	.N61_OUT AT %QB244 : ST_PSX_VALVE_OUT;	(*  ~ {LinkedWith:TIID^CAN 1 (BOW) ^PSX 61 (MF04)^RxPDO 1^Outputs^Device control word;TIID^CAN 1 (BOW) ^PSX 61 (MF04)^RxPDO 1^Outputs^vpoc_set_point_Value} *)
	.N64_OUT AT %QB248 : ST_PSX_VALVE_OUT;	(*  ~ {LinkedWith:TIID^CAN 1 (BOW) ^PSX 64 (MF04)^RxPDO 1^Outputs^Device control word;TIID^CAN 1 (BOW) ^PSX 64 (MF04)^RxPDO 1^Outputs^vpoc_set_point_Value} *)
	.EV4801 AT %QX696.0 : BOOL;
	.EV4802 AT %QX696.1 : BOOL;
	.EV4803 AT %QX696.2 : BOOL;
	.EV4804 AT %QX696.3 : BOOL;
	.N102_IN AT %IB502 : WORD;	(*  ~ {LinkedWith:TIID^CAN 4 (PANEL)^Box 102 (K-tronic CANopen Cariboni)^TxPDO 1^Entradas^Inputs} *)
	.N103_IN AT %IB504 : WORD;	(*  ~ {LinkedWith:TIID^CAN 4 (PANEL)^Box 103 (K-tronic CANopen Cariboni)^TxPDO 1^Entradas^Inputs} *)
	.N104_IN AT %IB506 : WORD;	(*  ~ {LinkedWith:TIID^CAN 4 (PANEL)^Box 104 (K-tronic CANopen Cariboni)^TxPDO 1^Entradas^Inputs} *)
	.N105_IN AT %IB508 : WORD;	(*  ~ {LinkedWith:TIID^CAN 4 (PANEL)^Box 105 (K-tronic CANopen Cariboni)^TxPDO 1^Entradas^Inputs} *)
	.N106_IN AT %IB510 : WORD;	(*  ~ {LinkedWith:TIID^CAN 4 (PANEL)^Box 106 (K-tronic CANopen Cariboni)^TxPDO 1^Entradas^Inputs} *)
	.N107_IN AT %IB512 : WORD;	(*  ~ {LinkedWith:TIID^CAN 4 (PANEL)^Box 107 (K-tronic CANopen Cariboni)^TxPDO 1^Entradas^Inputs} *)
	.N108_IN AT %IB514 : WORD;	(*  ~ {LinkedWith:TIID^CAN 4 (PANEL)^Box 108 (K-tronic CANopen Cariboni)^TxPDO 1^Entradas^Inputs} *)
	.N109_IN AT %IB516 : WORD;	(*  ~ {LinkedWith:TIID^CAN 4 (PANEL)^Box 109 (K-tronic CANopen Cariboni)^TxPDO 1^Entradas^Inputs} *)
	.N110_IN AT %IB518 : WORD;	(*  ~ {LinkedWith:TIID^CAN 4 (PANEL)^Box 110 (K-tronic CANopen Cariboni)^TxPDO 1^Entradas^Inputs} *)
	.N111_IN AT %IB520 : WORD;	(*  ~ {LinkedWith:TIID^CAN 4 (PANEL)^Box 111 (K-tronic CANopen Cariboni)^TxPDO 1^Entradas^Inputs} *)
	.N112_IN AT %IB522 : WORD;	(*  ~ {LinkedWith:TIID^CAN 4 (PANEL)^Box 112 (K-tronic CANopen Cariboni)^TxPDO 1^Entradas^Inputs} *)
	.N113_IN AT %IB524 : WORD;	(*  ~ {LinkedWith:TIID^CAN 4 (PANEL)^Box 113 (K-tronic CANopen Cariboni)^TxPDO 1^Entradas^Inputs} *)
	.N114_IN AT %IB526 : WORD;	(*  ~ {LinkedWith:TIID^CAN 4 (PANEL)^Box 114 (K-tronic CANopen Cariboni)^TxPDO 1^Entradas^Inputs} *)
	.N115_IN AT %IB528 : WORD;	(*  ~ {LinkedWith:TIID^CAN 4 (PANEL)^Box 115 (K-tronic CANopen Cariboni)^TxPDO 1^Entradas^Inputs} *)
	.N116_IN AT %IB530 : WORD;	(*  ~ {LinkedWith:TIID^CAN 4 (PANEL)^Box 116 (K-tronic CANopen Cariboni)^TxPDO 1^Entradas^Inputs} *)
	.N117_IN AT %IB532 : WORD;	(*  ~ {LinkedWith:TIID^CAN 4 (PANEL)^Box 117 (K-tronic CANopen Cariboni)^TxPDO 1^Entradas^Inputs} *)
	.N118_IN AT %IB534 : WORD;	(*  ~ {LinkedWith:TIID^CAN 4 (PANEL)^Box 118 (K-tronic CANopen Cariboni)^TxPDO 1^Entradas^Inputs} *)
	.N119_IN AT %IB536 : WORD;	(*  ~ {LinkedWith:TIID^CAN 4 (PANEL)^Box 119 (K-tronic CANopen Cariboni)^TxPDO 1^Entradas^Inputs} *)
	.N120_IN AT %IB744 : WORD;	(*  ~ {LinkedWith:TIID^CAN 4 (PANEL)^Box 120 (bLink)^TxPDO 1^Entradas^IN} *)
	.N121_IN AT %IB746 : WORD;	(*  ~ {LinkedWith:TIID^CAN 4 (PANEL)^Box 121 (bLink)^TxPDO 1^Entradas^IN} *)
	.N102_OUT AT %QB252 : WORD;	(*  ~ {LinkedWith:TIID^CAN 4 (PANEL)^Box 102 (K-tronic CANopen Cariboni)^RxPDO 1^Salidas^Outputs} *)
	.N103_OUT AT %QB254 : WORD;	(*  ~ {LinkedWith:TIID^CAN 4 (PANEL)^Box 103 (K-tronic CANopen Cariboni)^RxPDO 1^Salidas^Outputs} *)
	.N104_OUT AT %QB256 : WORD;	(*  ~ {LinkedWith:TIID^CAN 4 (PANEL)^Box 104 (K-tronic CANopen Cariboni)^RxPDO 1^Salidas^Outputs} *)
	.N105_OUT AT %QB258 : WORD;	(*  ~ {LinkedWith:TIID^CAN 4 (PANEL)^Box 105 (K-tronic CANopen Cariboni)^RxPDO 1^Salidas^Outputs} *)
	.N106_OUT AT %QB260 : WORD;	(*  ~ {LinkedWith:TIID^CAN 4 (PANEL)^Box 106 (K-tronic CANopen Cariboni)^RxPDO 1^Salidas^Outputs} *)
	.N107_OUT AT %QB262 : WORD;	(*  ~ {LinkedWith:TIID^CAN 4 (PANEL)^Box 107 (K-tronic CANopen Cariboni)^RxPDO 1^Salidas^Outputs} *)
	.N108_OUT AT %QB264 : WORD;	(*  ~ {LinkedWith:TIID^CAN 4 (PANEL)^Box 108 (K-tronic CANopen Cariboni)^RxPDO 1^Salidas^Outputs} *)
	.N109_OUT AT %QB266 : WORD;	(*  ~ {LinkedWith:TIID^CAN 4 (PANEL)^Box 109 (K-tronic CANopen Cariboni)^RxPDO 1^Salidas^Outputs} *)
	.N110_OUT AT %QB268 : WORD;	(*  ~ {LinkedWith:TIID^CAN 4 (PANEL)^Box 110 (K-tronic CANopen Cariboni)^RxPDO 1^Salidas^Outputs} *)
	.N111_OUT AT %QB270 : WORD;	(*  ~ {LinkedWith:TIID^CAN 4 (PANEL)^Box 111 (K-tronic CANopen Cariboni)^RxPDO 1^Salidas^Outputs} *)
	.N112_OUT AT %QB272 : WORD;	(*  ~ {LinkedWith:TIID^CAN 4 (PANEL)^Box 112 (K-tronic CANopen Cariboni)^RxPDO 1^Salidas^Outputs} *)
	.N113_OUT AT %QB274 : WORD;	(*  ~ {LinkedWith:TIID^CAN 4 (PANEL)^Box 113 (K-tronic CANopen Cariboni)^RxPDO 1^Salidas^Outputs} *)
	.N114_OUT AT %QB276 : WORD;	(*  ~ {LinkedWith:TIID^CAN 4 (PANEL)^Box 114 (K-tronic CANopen Cariboni)^RxPDO 1^Salidas^Outputs} *)
	.N115_OUT AT %QB278 : WORD;	(*  ~ {LinkedWith:TIID^CAN 4 (PANEL)^Box 115 (K-tronic CANopen Cariboni)^RxPDO 1^Salidas^Outputs} *)
	.N116_OUT AT %QB280 : WORD;	(*  ~ {LinkedWith:TIID^CAN 4 (PANEL)^Box 116 (K-tronic CANopen Cariboni)^RxPDO 1^Salidas^Outputs} *)
	.N117_OUT AT %QB282 : WORD;	(*  ~ {LinkedWith:TIID^CAN 4 (PANEL)^Box 117 (K-tronic CANopen Cariboni)^RxPDO 1^Salidas^Outputs} *)
	.N118_OUT AT %QB284 : WORD;	(*  ~ {LinkedWith:TIID^CAN 4 (PANEL)^Box 118 (K-tronic CANopen Cariboni)^RxPDO 1^Salidas^Outputs} *)
	.N119_OUT AT %QB286 : WORD;	(*  ~ {LinkedWith:TIID^CAN 4 (PANEL)^Box 119 (K-tronic CANopen Cariboni)^RxPDO 1^Salidas^Outputs} *)
	.N120_LED_R AT %QB664 : WORD;	(*  ~ {LinkedWith:TIID^CAN 4 (PANEL)^Box 120 (bLink)^RxPDO 1^Salidas^ON_RED} *)
	.N120_LED_G AT %QB666 : WORD;	(*  ~ {LinkedWith:TIID^CAN 4 (PANEL)^Box 120 (bLink)^RxPDO 1^Salidas^ON_GREEN} *)
	.N120_LED_B AT %QB668 : WORD;	(*  ~ {LinkedWith:TIID^CAN 4 (PANEL)^Box 120 (bLink)^RxPDO 1^Salidas^ON_BLUE} *)
	.N121_LED_R AT %QB670 : WORD;	(*  ~ {LinkedWith:TIID^CAN 4 (PANEL)^Box 121 (bLink)^RxPDO 1^Salidas^ON_RED} *)
	.N121_LED_G AT %QB672 : WORD;	(*  ~ {LinkedWith:TIID^CAN 4 (PANEL)^Box 121 (bLink)^RxPDO 1^Salidas^ON_GREEN} *)
	.N121_LED_B AT %QB674 : WORD;	(*  ~ {LinkedWith:TIID^CAN 4 (PANEL)^Box 121 (bLink)^RxPDO 1^Salidas^ON_BLUE} *)
	.N102_BLINK AT %QB288 : WORD;	(*  ~ {LinkedWith:TIID^CAN 4 (PANEL)^Box 102 (K-tronic CANopen Cariboni)^RxPDO 1^Salidas^BlinkOut} *)
	.N103_BLINK AT %QB290 : WORD;	(*  ~ {LinkedWith:TIID^CAN 4 (PANEL)^Box 103 (K-tronic CANopen Cariboni)^RxPDO 1^Salidas^BlinkOut} *)
	.N104_BLINK AT %QB292 : WORD;	(*  ~ {LinkedWith:TIID^CAN 4 (PANEL)^Box 104 (K-tronic CANopen Cariboni)^RxPDO 1^Salidas^BlinkOut} *)
	.N105_BLINK AT %QB294 : WORD;	(*  ~ {LinkedWith:TIID^CAN 4 (PANEL)^Box 105 (K-tronic CANopen Cariboni)^RxPDO 1^Salidas^BlinkOut} *)
	.N106_BLINK AT %QB296 : WORD;	(*  ~ {LinkedWith:TIID^CAN 4 (PANEL)^Box 106 (K-tronic CANopen Cariboni)^RxPDO 1^Salidas^BlinkOut} *)
	.N107_BLINK AT %QB298 : WORD;	(*  ~ {LinkedWith:TIID^CAN 4 (PANEL)^Box 107 (K-tronic CANopen Cariboni)^RxPDO 1^Salidas^BlinkOut} *)
	.N108_BLINK AT %QB300 : WORD;	(*  ~ {LinkedWith:TIID^CAN 4 (PANEL)^Box 108 (K-tronic CANopen Cariboni)^RxPDO 1^Salidas^BlinkOut} *)
	.N109_BLINK AT %QB302 : WORD;	(*  ~ {LinkedWith:TIID^CAN 4 (PANEL)^Box 109 (K-tronic CANopen Cariboni)^RxPDO 1^Salidas^BlinkOut} *)
	.N110_BLINK AT %QB304 : WORD;	(*  ~ {LinkedWith:TIID^CAN 4 (PANEL)^Box 110 (K-tronic CANopen Cariboni)^RxPDO 1^Salidas^BlinkOut} *)
	.N111_BLINK AT %QB306 : WORD;	(*  ~ {LinkedWith:TIID^CAN 4 (PANEL)^Box 111 (K-tronic CANopen Cariboni)^RxPDO 1^Salidas^BlinkOut} *)
	.N112_BLINK AT %QB308 : WORD;	(*  ~ {LinkedWith:TIID^CAN 4 (PANEL)^Box 112 (K-tronic CANopen Cariboni)^RxPDO 1^Salidas^BlinkOut} *)
	.N113_BLINK AT %QB310 : WORD;	(*  ~ {LinkedWith:TIID^CAN 4 (PANEL)^Box 113 (K-tronic CANopen Cariboni)^RxPDO 1^Salidas^BlinkOut} *)
	.N114_BLINK AT %QB312 : WORD;	(*  ~ {LinkedWith:TIID^CAN 4 (PANEL)^Box 114 (K-tronic CANopen Cariboni)^RxPDO 1^Salidas^BlinkOut} *)
	.N115_BLINK AT %QB314 : WORD;	(*  ~ {LinkedWith:TIID^CAN 4 (PANEL)^Box 115 (K-tronic CANopen Cariboni)^RxPDO 1^Salidas^BlinkOut} *)
	.N116_BLINK AT %QB316 : WORD;	(*  ~ {LinkedWith:TIID^CAN 4 (PANEL)^Box 116 (K-tronic CANopen Cariboni)^RxPDO 1^Salidas^BlinkOut} *)
	.N117_BLINK AT %QB318 : WORD;	(*  ~ {LinkedWith:TIID^CAN 4 (PANEL)^Box 117 (K-tronic CANopen Cariboni)^RxPDO 1^Salidas^BlinkOut} *)
	.N118_BLINK AT %QB320 : WORD;	(*  ~ {LinkedWith:TIID^CAN 4 (PANEL)^Box 118 (K-tronic CANopen Cariboni)^RxPDO 1^Salidas^BlinkOut} *)
	.N119_BLINK AT %QB322 : WORD;	(*  ~ {LinkedWith:TIID^CAN 4 (PANEL)^Box 119 (K-tronic CANopen Cariboni)^RxPDO 1^Salidas^BlinkOut} *)
	.N120_BLINK_R AT %QB676 : WORD;	(*  ~ {LinkedWith:TIID^CAN 4 (PANEL)^Box 120 (bLink)^RxPDO 2^Salidas^BLINK_RED} *)
	.N120_BLINK_G AT %QB678 : WORD;	(*  ~ {LinkedWith:TIID^CAN 4 (PANEL)^Box 120 (bLink)^RxPDO 2^Salidas^BLINK_GREEN} *)
	.N120_BLINK_B AT %QB680 : WORD;	(*  ~ {LinkedWith:TIID^CAN 4 (PANEL)^Box 120 (bLink)^RxPDO 2^Salidas^BLINK_BLUE} *)
	.N121_BLINK_R AT %QB682 : WORD;	(*  ~ {LinkedWith:TIID^CAN 4 (PANEL)^Box 121 (bLink)^RxPDO 2^Salidas^BLINK_RED} *)
	.N121_BLINK_G AT %QB684 : WORD;	(*  ~ {LinkedWith:TIID^CAN 4 (PANEL)^Box 121 (bLink)^RxPDO 2^Salidas^BLINK_GREEN} *)
	.N121_BLINK_B AT %QB686 : WORD;	(*  ~ {LinkedWith:TIID^CAN 4 (PANEL)^Box 121 (bLink)^RxPDO 2^Salidas^BLINK_BLUE} *)
	.N102_BTIME AT %QB324 : BYTE;	(*  ~ {LinkedWith:TIID^CAN 4 (PANEL)^Box 102 (K-tronic CANopen Cariboni)^RxPDO 1^Salidas^BlinkTime} *)
	.N103_BTIME AT %QB325 : BYTE;	(*  ~ {LinkedWith:TIID^CAN 4 (PANEL)^Box 103 (K-tronic CANopen Cariboni)^RxPDO 1^Salidas^BlinkTime} *)
	.N104_BTIME AT %QB326 : BYTE;	(*  ~ {LinkedWith:TIID^CAN 4 (PANEL)^Box 104 (K-tronic CANopen Cariboni)^RxPDO 1^Salidas^BlinkTime} *)
	.N105_BTIME AT %QB327 : BYTE;	(*  ~ {LinkedWith:TIID^CAN 4 (PANEL)^Box 105 (K-tronic CANopen Cariboni)^RxPDO 1^Salidas^BlinkTime} *)
	.N106_BTIME AT %QB328 : BYTE;	(*  ~ {LinkedWith:TIID^CAN 4 (PANEL)^Box 106 (K-tronic CANopen Cariboni)^RxPDO 1^Salidas^BlinkTime} *)
	.N107_BTIME AT %QB329 : BYTE;	(*  ~ {LinkedWith:TIID^CAN 4 (PANEL)^Box 107 (K-tronic CANopen Cariboni)^RxPDO 1^Salidas^BlinkTime} *)
	.N108_BTIME AT %QB330 : BYTE;	(*  ~ {LinkedWith:TIID^CAN 4 (PANEL)^Box 108 (K-tronic CANopen Cariboni)^RxPDO 1^Salidas^BlinkTime} *)
	.N109_BTIME AT %QB331 : BYTE;	(*  ~ {LinkedWith:TIID^CAN 4 (PANEL)^Box 109 (K-tronic CANopen Cariboni)^RxPDO 1^Salidas^BlinkTime} *)
	.N110_BTIME AT %QB332 : BYTE;	(*  ~ {LinkedWith:TIID^CAN 4 (PANEL)^Box 110 (K-tronic CANopen Cariboni)^RxPDO 1^Salidas^BlinkTime} *)
	.N111_BTIME AT %QB333 : BYTE;	(*  ~ {LinkedWith:TIID^CAN 4 (PANEL)^Box 111 (K-tronic CANopen Cariboni)^RxPDO 1^Salidas^BlinkTime} *)
	.N112_BTIME AT %QB334 : BYTE;	(*  ~ {LinkedWith:TIID^CAN 4 (PANEL)^Box 112 (K-tronic CANopen Cariboni)^RxPDO 1^Salidas^BlinkTime} *)
	.N113_BTIME AT %QB335 : BYTE;	(*  ~ {LinkedWith:TIID^CAN 4 (PANEL)^Box 113 (K-tronic CANopen Cariboni)^RxPDO 1^Salidas^BlinkTime} *)
	.N114_BTIME AT %QB336 : BYTE;	(*  ~ {LinkedWith:TIID^CAN 4 (PANEL)^Box 114 (K-tronic CANopen Cariboni)^RxPDO 1^Salidas^BlinkTime} *)
	.N115_BTIME AT %QB337 : BYTE;	(*  ~ {LinkedWith:TIID^CAN 4 (PANEL)^Box 115 (K-tronic CANopen Cariboni)^RxPDO 1^Salidas^BlinkTime} *)
	.N116_BTIME AT %QB338 : BYTE;	(*  ~ {LinkedWith:TIID^CAN 4 (PANEL)^Box 116 (K-tronic CANopen Cariboni)^RxPDO 1^Salidas^BlinkTime} *)
	.N117_BTIME AT %QB339 : BYTE;	(*  ~ {LinkedWith:TIID^CAN 4 (PANEL)^Box 117 (K-tronic CANopen Cariboni)^RxPDO 1^Salidas^BlinkTime} *)
	.N118_BTIME AT %QB340 : BYTE;	(*  ~ {LinkedWith:TIID^CAN 4 (PANEL)^Box 118 (K-tronic CANopen Cariboni)^RxPDO 1^Salidas^BlinkTime} *)
	.N119_BTIME AT %QB341 : BYTE;	(*  ~ {LinkedWith:TIID^CAN 4 (PANEL)^Box 119 (K-tronic CANopen Cariboni)^RxPDO 1^Salidas^BlinkTime} *)
	.N102_DIMMER AT %QB342 : WORD;	(*  ~ {LinkedWith:TIID^CAN 4 (PANEL)^Box 102 (K-tronic CANopen Cariboni)^RxPDO 3^Salidas^Dimmer1} *)
	.N103_DIMMER AT %QB344 : WORD;	(*  ~ {LinkedWith:TIID^CAN 4 (PANEL)^Box 103 (K-tronic CANopen Cariboni)^RxPDO 3^Salidas^Dimmer1} *)
	.N104_DIMMER AT %QB346 : WORD;	(*  ~ {LinkedWith:TIID^CAN 4 (PANEL)^Box 104 (K-tronic CANopen Cariboni)^RxPDO 3^Salidas^Dimmer1} *)
	.N105_DIMMER AT %QB348 : WORD;	(*  ~ {LinkedWith:TIID^CAN 4 (PANEL)^Box 105 (K-tronic CANopen Cariboni)^RxPDO 3^Salidas^Dimmer1} *)
	.N106_DIMMER AT %QB350 : WORD;	(*  ~ {LinkedWith:TIID^CAN 4 (PANEL)^Box 106 (K-tronic CANopen Cariboni)^RxPDO 3^Salidas^Dimmer1} *)
	.N107_DIMMER AT %QB352 : WORD;	(*  ~ {LinkedWith:TIID^CAN 4 (PANEL)^Box 107 (K-tronic CANopen Cariboni)^RxPDO 3^Salidas^Dimmer1} *)
	.N108_DIMMER AT %QB354 : WORD;	(*  ~ {LinkedWith:TIID^CAN 4 (PANEL)^Box 108 (K-tronic CANopen Cariboni)^RxPDO 3^Salidas^Dimmer1} *)
	.N109_DIMMER AT %QB356 : WORD;	(*  ~ {LinkedWith:TIID^CAN 4 (PANEL)^Box 109 (K-tronic CANopen Cariboni)^RxPDO 3^Salidas^Dimmer1} *)
	.N110_DIMMER AT %QB358 : WORD;	(*  ~ {LinkedWith:TIID^CAN 4 (PANEL)^Box 110 (K-tronic CANopen Cariboni)^RxPDO 3^Salidas^Dimmer1} *)
	.N111_DIMMER AT %QB360 : WORD;	(*  ~ {LinkedWith:TIID^CAN 4 (PANEL)^Box 111 (K-tronic CANopen Cariboni)^RxPDO 3^Salidas^Dimmer1} *)
	.N112_DIMMER AT %QB362 : WORD;	(*  ~ {LinkedWith:TIID^CAN 4 (PANEL)^Box 112 (K-tronic CANopen Cariboni)^RxPDO 3^Salidas^Dimmer1} *)
	.N113_DIMMER AT %QB364 : WORD;	(*  ~ {LinkedWith:TIID^CAN 4 (PANEL)^Box 113 (K-tronic CANopen Cariboni)^RxPDO 3^Salidas^Dimmer1} *)
	.N114_DIMMER AT %QB366 : WORD;	(*  ~ {LinkedWith:TIID^CAN 4 (PANEL)^Box 114 (K-tronic CANopen Cariboni)^RxPDO 3^Salidas^Dimmer1} *)
	.N115_DIMMER AT %QB368 : WORD;	(*  ~ {LinkedWith:TIID^CAN 4 (PANEL)^Box 115 (K-tronic CANopen Cariboni)^RxPDO 3^Salidas^Dimmer1} *)
	.N116_DIMMER AT %QB370 : WORD;	(*  ~ {LinkedWith:TIID^CAN 4 (PANEL)^Box 116 (K-tronic CANopen Cariboni)^RxPDO 3^Salidas^Dimmer1} *)
	.N117_DIMMER AT %QB372 : WORD;	(*  ~ {LinkedWith:TIID^CAN 4 (PANEL)^Box 117 (K-tronic CANopen Cariboni)^RxPDO 3^Salidas^Dimmer1} *)
	.N118_DIMMER AT %QB374 : WORD;	(*  ~ {LinkedWith:TIID^CAN 4 (PANEL)^Box 118 (K-tronic CANopen Cariboni)^RxPDO 3^Salidas^Dimmer1} *)
	.N119_DIMMER AT %QB376 : WORD;	(*  ~ {LinkedWith:TIID^CAN 4 (PANEL)^Box 119 (K-tronic CANopen Cariboni)^RxPDO 3^Salidas^Dimmer1} *)
	.N120_LED_Bright AT %QB688 : BYTE;	(*  ~ {LinkedWith:TIID^CAN 4 (PANEL)^Box 120 (bLink)^RxPDO 3^Salidas^LED_BRIGHT} *)
	.N121_LED_Bright AT %QB689 : BYTE;	(*  ~ {LinkedWith:TIID^CAN 4 (PANEL)^Box 121 (bLink)^RxPDO 3^Salidas^LED_BRIGHT} *)
	.N120_BL_Bright AT %QB690 : BYTE;	(*  ~ {LinkedWith:TIID^CAN 4 (PANEL)^Box 120 (bLink)^RxPDO 4^Salidas^BL_BRIGHT} *)
	.N121_BL_Bright AT %QB691 : BYTE;	(*  ~ {LinkedWith:TIID^CAN 4 (PANEL)^Box 121 (bLink)^RxPDO 4^Salidas^BL_BRIGHT} *)
	.N120_BL_Color AT %QB692 : BYTE;	(*  ~ {LinkedWith:TIID^CAN 4 (PANEL)^Box 120 (bLink)^RxPDO 4^Salidas^BL_COLOR} *)
	.N121_BL_Color AT %QB693 : BYTE;	(*  ~ {LinkedWith:TIID^CAN 4 (PANEL)^Box 121 (bLink)^RxPDO 4^Salidas^BL_COLOR} *)
	.CLM8_LED1 AT %QB520 : BYTE;	(*  ~ {LinkedWith:TIID^CAN 4 (PANEL)^Box 10 (CLM8)^COB 0x20A^Salidas^LED} *)
	.CLM8_LED2 AT %QB521 : BYTE;	(*  ~ {LinkedWith:TIID^CAN 4 (PANEL)^Box 10 (CLM8)^COB 0x20B^Salidas^LED} *)
	.CLM8_COLOR1 AT %QB524 : UDINT;	(*  ~ {LinkedWith:TIID^CAN 4 (PANEL)^Box 10 (CLM8)^COB 0x20A^Salidas^COLORS} *)
	.CLM8_COLOR2 AT %QB528 : UDINT;	(*  ~ {LinkedWith:TIID^CAN 4 (PANEL)^Box 10 (CLM8)^COB 0x20B^Salidas^COLORS} *)
	.CLM8_BRIGHT AT %QB532 : BYTE;	(*  ~ {LinkedWith:TIID^CAN 4 (PANEL)^Box 10 (CLM8)^COB 0x72F^Salidas^Brightness} *)
	.N10_DI0 AT %IX768.0 : BOOL;	(*  ~ {LinkedWith:TIID^CAN 5 (EL6751)^N10 (IP1001-510)^Term 1^Channel 1^Input} *)
	.N10_DI1 AT %IX768.1 : BOOL;	(*  ~ {LinkedWith:TIID^CAN 5 (EL6751)^N10 (IP1001-510)^Term 1^Channel 2^Input} *)
	.N10_DI2 AT %IX768.2 : BOOL;	(*  ~ {LinkedWith:TIID^CAN 5 (EL6751)^N10 (IP1001-510)^Term 1^Channel 3^Input} *)
	.N10_DI3 AT %IX768.3 : BOOL;	(*  ~ {LinkedWith:TIID^CAN 5 (EL6751)^N10 (IP1001-510)^Term 1^Channel 4^Input} *)
	.N10_DI4 AT %IX768.4 : BOOL;	(*  ~ {LinkedWith:TIID^CAN 5 (EL6751)^N10 (IP1001-510)^Term 1^Channel 5^Input} *)
	.N10_DI5 AT %IX768.5 : BOOL;	(*  ~ {LinkedWith:TIID^CAN 5 (EL6751)^N10 (IP1001-510)^Term 1^Channel 6^Input} *)
	.N10_DI6 AT %IX768.6 : BOOL;	(*  ~ {LinkedWith:TIID^CAN 5 (EL6751)^N10 (IP1001-510)^Term 1^Channel 7^Input} *)
	.N10_DI7 AT %IX768.7 : BOOL;	(*  ~ {LinkedWith:TIID^CAN 5 (EL6751)^N10 (IP1001-510)^Term 1^Channel 8^Input} *)
	.N11_DI0 AT %IX769.0 : BOOL;	(*  ~ {LinkedWith:TIID^CAN 5 (EL6751)^N11 (IP1001-510)^Term 1^Channel 1^Input} *)
	.N11_DI1 AT %IX769.1 : BOOL;	(*  ~ {LinkedWith:TIID^CAN 5 (EL6751)^N11 (IP1001-510)^Term 1^Channel 2^Input} *)
	.N11_DI2 AT %IX769.2 : BOOL;	(*  ~ {LinkedWith:TIID^CAN 5 (EL6751)^N11 (IP1001-510)^Term 1^Channel 3^Input} *)
	.N11_DI3 AT %IX769.3 : BOOL;	(*  ~ {LinkedWith:TIID^CAN 5 (EL6751)^N11 (IP1001-510)^Term 1^Channel 4^Input} *)
	.N11_DI4 AT %IX769.4 : BOOL;	(*  ~ {LinkedWith:TIID^CAN 5 (EL6751)^N11 (IP1001-510)^Term 1^Channel 5^Input} *)
	.N11_DI5 AT %IX769.5 : BOOL;	(*  ~ {LinkedWith:TIID^CAN 5 (EL6751)^N11 (IP1001-510)^Term 1^Channel 6^Input} *)
	.N11_DI6 AT %IX769.6 : BOOL;	(*  ~ {LinkedWith:TIID^CAN 5 (EL6751)^N11 (IP1001-510)^Term 1^Channel 7^Input} *)
	.N11_DI7 AT %IX769.7 : BOOL;	(*  ~ {LinkedWith:TIID^CAN 5 (EL6751)^N11 (IP1001-510)^Term 1^Channel 8^Input} *)
	.N12_DI0 AT %IX770.0 : BOOL;	(*  ~ {LinkedWith:TIID^CAN 5 (EL6751)^N12 (IP1001-510)^Term 1^Channel 1^Input} *)
	.N12_DI1 AT %IX770.1 : BOOL;	(*  ~ {LinkedWith:TIID^CAN 5 (EL6751)^N12 (IP1001-510)^Term 1^Channel 2^Input} *)
	.N12_DI2 AT %IX770.2 : BOOL;	(*  ~ {LinkedWith:TIID^CAN 5 (EL6751)^N12 (IP1001-510)^Term 1^Channel 3^Input} *)
	.N12_DI3 AT %IX770.3 : BOOL;	(*  ~ {LinkedWith:TIID^CAN 5 (EL6751)^N12 (IP1001-510)^Term 1^Channel 4^Input} *)
	.N12_DI4 AT %IX770.4 : BOOL;	(*  ~ {LinkedWith:TIID^CAN 5 (EL6751)^N12 (IP1001-510)^Term 1^Channel 5^Input} *)
	.N12_DI5 AT %IX770.5 : BOOL;	(*  ~ {LinkedWith:TIID^CAN 5 (EL6751)^N12 (IP1001-510)^Term 1^Channel 6^Input} *)
	.N12_DI6 AT %IX770.6 : BOOL;	(*  ~ {LinkedWith:TIID^CAN 5 (EL6751)^N12 (IP1001-510)^Term 1^Channel 7^Input} *)
	.N12_DI7 AT %IX770.7 : BOOL;	(*  ~ {LinkedWith:TIID^CAN 5 (EL6751)^N12 (IP1001-510)^Term 1^Channel 8^Input} *)
	.N13_DI0 AT %IX771.0 : BOOL;	(*  ~ {LinkedWith:TIID^CAN 5 (EL6751)^N13 (IP1001-510)^Term 1^Channel 1^Input} *)
	.N13_DI1 AT %IX771.1 : BOOL;	(*  ~ {LinkedWith:TIID^CAN 5 (EL6751)^N13 (IP1001-510)^Term 1^Channel 2^Input} *)
	.N13_DI2 AT %IX771.2 : BOOL;	(*  ~ {LinkedWith:TIID^CAN 5 (EL6751)^N13 (IP1001-510)^Term 1^Channel 3^Input} *)
	.N13_DI3 AT %IX771.3 : BOOL;	(*  ~ {LinkedWith:TIID^CAN 5 (EL6751)^N13 (IP1001-510)^Term 1^Channel 4^Input} *)
	.N13_DI4 AT %IX771.4 : BOOL;	(*  ~ {LinkedWith:TIID^CAN 5 (EL6751)^N13 (IP1001-510)^Term 1^Channel 5^Input} *)
	.N13_DI5 AT %IX771.5 : BOOL;	(*  ~ {LinkedWith:TIID^CAN 5 (EL6751)^N13 (IP1001-510)^Term 1^Channel 6^Input} *)
	.N13_DI6 AT %IX771.6 : BOOL;	(*  ~ {LinkedWith:TIID^CAN 5 (EL6751)^N13 (IP1001-510)^Term 1^Channel 7^Input} *)
	.N13_DI7 AT %IX771.7 : BOOL;	(*  ~ {LinkedWith:TIID^CAN 5 (EL6751)^N13 (IP1001-510)^Term 1^Channel 8^Input} *)
	.N20_DI0 AT %IX772.0 : BOOL;	(*  ~ {LinkedWith:TIID^CAN 5 (EL6751)^N20 (IP1001-510)^Term 1^Channel 1^Input} *)
	.N20_DI1 AT %IX772.1 : BOOL;	(*  ~ {LinkedWith:TIID^CAN 5 (EL6751)^N20 (IP1001-510)^Term 1^Channel 2^Input} *)
	.N20_DI2 AT %IX772.2 : BOOL;	(*  ~ {LinkedWith:TIID^CAN 5 (EL6751)^N20 (IP1001-510)^Term 1^Channel 3^Input} *)
	.N20_DI3 AT %IX772.3 : BOOL;	(*  ~ {LinkedWith:TIID^CAN 5 (EL6751)^N20 (IP1001-510)^Term 1^Channel 4^Input} *)
	.N20_DI4 AT %IX772.4 : BOOL;	(*  ~ {LinkedWith:TIID^CAN 5 (EL6751)^N20 (IP1001-510)^Term 1^Channel 5^Input} *)
	.N20_DI5 AT %IX772.5 : BOOL;	(*  ~ {LinkedWith:TIID^CAN 5 (EL6751)^N20 (IP1001-510)^Term 1^Channel 6^Input} *)
	.N20_DI6 AT %IX772.6 : BOOL;	(*  ~ {LinkedWith:TIID^CAN 5 (EL6751)^N20 (IP1001-510)^Term 1^Channel 7^Input} *)
	.N20_DI7 AT %IX772.7 : BOOL;	(*  ~ {LinkedWith:TIID^CAN 5 (EL6751)^N20 (IP1001-510)^Term 1^Channel 8^Input} *)
	.N20_NodeState AT %IB592 : USINT;	(*  ~ {LinkedWith:TIID^CAN 1 (BOW) ^Box 20 (MF06)^Entradas^NodeState} *)
	.N21_NodeState AT %IB593 : USINT;	(*  ~ {LinkedWith:TIID^CAN 1 (BOW) ^Box 21 (MF07/MF11)^Entradas^NodeState} *)
	.N22_NodeState AT %IB594 : USINT;	(*  ~ {LinkedWith:TIID^CAN 1 (BOW) ^Box 22 (MF07)^Entradas^NodeState} *)
	.N23_NodeState AT %IB595 : USINT;	(*  ~ {LinkedWith:TIID^CAN 2 (STERN)^Box 23 (MF08)^Entradas^NodeState} *)
	.N24_NodeState AT %IB596 : USINT;	(*  ~ {LinkedWith:TIID^CAN 2 (STERN)^Box 24 (MF12A)^Entradas^NodeState} *)
	.N25_NodeState AT %IB597 : USINT;	(*  ~ {LinkedWith:TIID^CAN 2 (STERN)^Box 25 (MF12B)^Entradas^NodeState} *)
	.N26_NodeState AT %IB598 : USINT;	(*  ~ {LinkedWith:TIID^CAN 2 (STERN)^Box 26 (MF25)^Entradas^NodeState} *)
	.N27_NodeState AT %IB599 : USINT;	(*  ~ {LinkedWith:TIID^CAN 2 (STERN)^Box 27 (MF22)^Entradas^NodeState} *)
	.N28_NodeState AT %IB600 : USINT;	(*  ~ {LinkedWith:TIID^CAN 2 (STERN)^Box 28 (MF21)^Entradas^NodeState} *)
	.N29_NodeState AT %IB601 : USINT;	(*  ~ {LinkedWith:TIID^CAN 2 (STERN)^Box 29 (MF24)^Entradas^NodeState} *)
	.N30_NodeState AT %IB602 : USINT;	(*  ~ {LinkedWith:TIID^CAN 2 (STERN)^Box 30 (MF23)^Entradas^NodeState} *)
	.N31_NodeState AT %IB603 : USINT;	(*  ~ {LinkedWith:TIID^CAN 2 (STERN)^Box 31 (MF20)^Entradas^NodeState} *)
	.N32_NodeState AT %IB604 : USINT;	(*  ~ {LinkedWith:TIID^CAN 2 (STERN)^Box 32 (MF19)^Entradas^NodeState} *)
	.N33_NodeState AT %IB605 : USINT;	(*  ~ {LinkedWith:TIID^CAN 2 (STERN)^Box 33 (MF13 Traveller)^Entradas^NodeState} *)
	.N34_NodeState AT %IB606 : USINT;	(*  ~ {LinkedWith:TIID^CAN 2 (STERN)^Box 34 (MF16)^Entradas^NodeState} *)
	.N35_NodeState AT %IB607 : USINT;	(*  ~ {LinkedWith:TIID^CAN 2 (STERN)^Box 35 (MF09)^Entradas^NodeState} *)
	.N36_NodeState AT %IB608 : USINT;	(*  ~ {LinkedWith:TIID^CAN 1 (BOW) ^Box 36 (Tank)^Entradas^NodeState} *)
	.N37_NodeState AT %IB609 : USINT;	(*  ~ {LinkedWith:TIID^CAN 1 (BOW) ^Box 37 (Tank)^Entradas^NodeState} *)
	.N38_NodeState AT %IB610 : USINT;	(*  ~ {LinkedWith:TIID^CAN 2 (STERN)^Box 38 (LIGHT)^Entradas^NodeState} *)
	.N39_NodeState AT %IB611 : USINT;	(*  ~ {LinkedWith:TIID^CAN 1 (BOW) ^Box 39 (MF10A Keel)^Entradas^NodeState} *)
	.N40_NodeState AT %IB612 : USINT;	(*  ~ {LinkedWith:TIID^CAN 1 (BOW) ^Box 40 (MF10B Keel)^Entradas^NodeState} *)
	.N41_NodeState AT %IB613 : USINT;	(*  ~ {LinkedWith:TIID^CAN 1 (BOW) ^Box 41 (MF05)^Entradas^NodeState} *)
	.N42_NodeState AT %IB614 : USINT;	(*  ~ {LinkedWith:TIID^CAN 1 (BOW) ^Box 42 (MF01 HP PP)^Entradas^NodeState} *)
	.N43_NodeState AT %IB615 : USINT;	(*  ~ {LinkedWith:TIID^CAN 1 (BOW) ^Box 43 (MF03A)^Entradas^NodeState} *)
	.N44_NodeState AT %IB616 : USINT;	(*  ~ {LinkedWith:TIID^CAN 1 (BOW) ^Box 44 (MF03B)^Entradas^NodeState} *)
	.N47_NodeState AT %IB706 : USINT;	(*  ~ {LinkedWith:TIID^CAN 2 (STERN)^Box 47 (MF11)^Entradas^NodeState} *)
	.N48_NodeState AT %IB764 : USINT;	(*  ~ {LinkedWith:TIID^CAN 1 (BOW) ^Box 48 (DGB Seal)^Entradas^NodeState} *)
	.N50_NodeState AT %IB617 : USINT;	(*  ~ {LinkedWith:TIID^CAN 2 (STERN)^PSX 50 (MF12)^Inputs^NodeState} *)
	.N51_NodeState AT %IB618 : USINT;	(*  ~ {LinkedWith:TIID^CAN 2 (STERN)^PSX 51 (MF12)^Inputs^NodeState} *)
	.N52_NodeState AT %IB619 : USINT;	(*  ~ {LinkedWith:TIID^CAN 2 (STERN)^PSX 52 (MF12)^Inputs^NodeState} *)
	.N53_NodeState AT %IB620 : USINT;	(*  ~ {LinkedWith:TIID^CAN 2 (STERN)^PSX 53 (MF12)^Inputs^NodeState} *)
	.N54_NodeState AT %IB621 : USINT;	(*  ~ {LinkedWith:TIID^CAN 2 (STERN)^PSX 54 (MF12)^Inputs^NodeState} *)
	.N55_NodeState AT %IB622 : USINT;	(*  ~ {LinkedWith:TIID^CAN 2 (STERN)^PSX 55 (MF12)^Inputs^NodeState} *)
	.N56_NodeState AT %IB623 : USINT;	(*  ~ {LinkedWith:TIID^CAN 2 (STERN)^PSX 56 (MF12)^Inputs^NodeState} *)
	.N57_NodeState AT %IB624 : USINT;	(*  ~ {LinkedWith:TIID^CAN 2 (STERN)^PSX 57 (MF12)^Inputs^NodeState} *)
	.N58_NodeState AT %IB625 : USINT;	(*  ~ {LinkedWith:TIID^CAN 2 (STERN)^PSX 58 (MF12)^Inputs^NodeState} *)
	.N59_NodeState AT %IB626 : USINT;	(*  ~ {LinkedWith:TIID^CAN 2 (STERN)^PSX 59 (MF12)^Inputs^NodeState} *)
	.N60_NodeState AT %IB627 : USINT;	(*  ~ {LinkedWith:TIID^CAN 1 (BOW) ^PSX 60 (MF04)^Inputs^NodeState} *)
	.N61_NodeState AT %IB628 : USINT;	(*  ~ {LinkedWith:TIID^CAN 1 (BOW) ^PSX 61 (MF04)^Inputs^NodeState} *)
	.N64_NodeState AT %IB629 : USINT;	(*  ~ {LinkedWith:TIID^CAN 1 (BOW) ^PSX 64 (MF04)^Inputs^NodeState} *)
	.N70_NodeState AT %IB630 : USINT;	(*  ~ {LinkedWith:TIID^CAN 2 (STERN)^PSX 70 (MF16)^Inputs^NodeState} *)
	.N71_NodeState AT %IB631 : USINT;	(*  ~ {LinkedWith:TIID^CAN 2 (STERN)^PSX 71 (MF16)^Inputs^NodeState} *)
	.N72_NodeState AT %IB632 : USINT;	(*  ~ {LinkedWith:TIID^CAN 2 (STERN)^PSX 72 (MF16)^Inputs^NodeState} *)
	.N73_NodeState AT %IB633 : USINT;	(*  ~ {LinkedWith:TIID^CAN 2 (STERN)^PSX 73 (MF16)^Inputs^NodeState} *)
	.N74_NodeState AT %IB634 : USINT;	(*  ~ {LinkedWith:TIID^CAN 2 (STERN)^PSX 74 (MF16)^Inputs^NodeState} *)
	.N102_NodeState AT %IB635 : USINT;	(*  ~ {LinkedWith:TIID^CAN 4 (PANEL)^Box 102 (K-tronic CANopen Cariboni)^Entradas^NodeState} *)
	.N103_NodeState AT %IB636 : USINT;	(*  ~ {LinkedWith:TIID^CAN 4 (PANEL)^Box 103 (K-tronic CANopen Cariboni)^Entradas^NodeState} *)
	.N104_NodeState AT %IB637 : USINT;	(*  ~ {LinkedWith:TIID^CAN 4 (PANEL)^Box 104 (K-tronic CANopen Cariboni)^Entradas^NodeState} *)
	.N105_NodeState AT %IB638 : USINT;	(*  ~ {LinkedWith:TIID^CAN 4 (PANEL)^Box 105 (K-tronic CANopen Cariboni)^Entradas^NodeState} *)
	.N106_NodeState AT %IB639 : USINT;	(*  ~ {LinkedWith:TIID^CAN 4 (PANEL)^Box 106 (K-tronic CANopen Cariboni)^Entradas^NodeState} *)
	.N107_NodeState AT %IB640 : USINT;	(*  ~ {LinkedWith:TIID^CAN 4 (PANEL)^Box 107 (K-tronic CANopen Cariboni)^Entradas^NodeState} *)
	.N108_NodeState AT %IB641 : USINT;	(*  ~ {LinkedWith:TIID^CAN 4 (PANEL)^Box 108 (K-tronic CANopen Cariboni)^Entradas^NodeState} *)
	.N109_NodeState AT %IB642 : USINT;	(*  ~ {LinkedWith:TIID^CAN 4 (PANEL)^Box 109 (K-tronic CANopen Cariboni)^Entradas^NodeState} *)
	.N110_NodeState AT %IB643 : USINT;	(*  ~ {LinkedWith:TIID^CAN 4 (PANEL)^Box 110 (K-tronic CANopen Cariboni)^Entradas^NodeState} *)
	.N111_NodeState AT %IB644 : USINT;	(*  ~ {LinkedWith:TIID^CAN 4 (PANEL)^Box 111 (K-tronic CANopen Cariboni)^Entradas^NodeState} *)
	.N112_NodeState AT %IB645 : USINT;	(*  ~ {LinkedWith:TIID^CAN 4 (PANEL)^Box 112 (K-tronic CANopen Cariboni)^Entradas^NodeState} *)
	.N113_NodeState AT %IB646 : USINT;	(*  ~ {LinkedWith:TIID^CAN 4 (PANEL)^Box 113 (K-tronic CANopen Cariboni)^Entradas^NodeState} *)
	.N114_NodeState AT %IB647 : USINT;	(*  ~ {LinkedWith:TIID^CAN 4 (PANEL)^Box 114 (K-tronic CANopen Cariboni)^Entradas^NodeState} *)
	.N115_NodeState AT %IB648 : USINT;	(*  ~ {LinkedWith:TIID^CAN 4 (PANEL)^Box 115 (K-tronic CANopen Cariboni)^Entradas^NodeState} *)
	.N116_NodeState AT %IB649 : USINT;	(*  ~ {LinkedWith:TIID^CAN 4 (PANEL)^Box 116 (K-tronic CANopen Cariboni)^Entradas^NodeState} *)
	.N117_NodeState AT %IB650 : USINT;	(*  ~ {LinkedWith:TIID^CAN 4 (PANEL)^Box 117 (K-tronic CANopen Cariboni)^Entradas^NodeState} *)
	.N118_NodeState AT %IB651 : USINT;	(*  ~ {LinkedWith:TIID^CAN 4 (PANEL)^Box 118 (K-tronic CANopen Cariboni)^Entradas^NodeState} *)
	.N119_NodeState AT %IB652 : USINT;	(*  ~ {LinkedWith:TIID^CAN 4 (PANEL)^Box 119 (K-tronic CANopen Cariboni)^Entradas^NodeState} *)
	.N120_NodeState AT %IB748 : USINT;	(*  ~ {LinkedWith:TIID^CAN 4 (PANEL)^Box 120 (bLink)^Entradas^NodeState} *)
	.N121_NodeState AT %IB749 : USINT;	(*  ~ {LinkedWith:TIID^CAN 4 (PANEL)^Box 121 (bLink)^Entradas^NodeState} *)
	.N10_NodeState AT %IB661 : USINT;	(*  ~ {LinkedWith:TIID^CAN 5 (EL6751)^N10 (IP1001-510)^Inputs^NodeState} *)
	.N11_NodeState AT %IB662 : USINT;	(*  ~ {LinkedWith:TIID^CAN 5 (EL6751)^N11 (IP1001-510)^Inputs^NodeState} *)
	.N12_NodeState AT %IB663 : USINT;	(*  ~ {LinkedWith:TIID^CAN 5 (EL6751)^N12 (IP1001-510)^Inputs^NodeState} *)
	.N13_NodeState AT %IB664 : USINT;	(*  ~ {LinkedWith:TIID^CAN 5 (EL6751)^N13 (IP1001-510)^Inputs^NodeState} *)
	.N20_2_NodeState AT %IB724 : USINT;	(*  ~ {LinkedWith:TIID^CAN 5 (EL6751)^N20 (IP1001-510)^Inputs^NodeState} *)
END_VAR

(* Data type *)
TYPE RxQueue_10 :
STRUCT
	TxCounter      : UINT;
	RxCounter      : UINT;
	NoOfRxMessages : UINT;
	RxMessages     : ARRAY [0..9] OF ARRAY[0..13] OF BYTE;
END_STRUCT
END_TYPE

(* Data type *)
TYPE ST_ALARM :
STRUCT
	AlLen  : REAL;
	AlCnt  : WORD;
	TimeInit : STRING;
	TimeEnd  : STRING;

	Alarm  : BOOL;
	Adver  : BOOL;
	Text   : STRING;

	AlInit : BOOL;
	AlEnd  : BOOL;
END_STRUCT
END_TYPE

(* Data type *)
TYPE ST_BOARD_CFG :
STRUCT
(*Targets*)
	TgtLS_P_In   : REAL;
	TgtLS_P_InR  : REAL;
	TgtLS_P_Mid  : REAL;
	TgtLS_P_OutR : REAL;
	TgtLS_P_Out  : REAL;

	TgtLS_S_In   : REAL;
	TgtLS_S_InR  : REAL;
	TgtLS_S_Mid  : REAL;
	TgtLS_S_OutR : REAL;
	TgtLS_S_Out  : REAL;

	TgtLS_P_Safe_Out : REAL;
	TgtLS_P_Safe_In  : REAL;

	TgtLS_S_Safe_Out : REAL;
	TgtLS_S_Safe_In  : REAL;

	LS_Dif_Tgt : REAL;
	LS_Dif_Max : REAL;
	LS_Dif_Min : REAL;

	LS_DB : REAL;

	P_Hyst_HP : REAL;
	P_Hyst_LP : REAL;
	P_Hyst_TM : REAL;	(*Seconds*)

(*Keel Limits*)
	Keel_P_Max : REAL;
	Keel_S_Min : REAL;

(*Valve Limits*)
	EVP_In_P_Min  : REAL;
	EVP_In_P_Max  : REAL;

	EVP_In_S_Min  : REAL;
	EVP_In_S_Max  : REAL;

	EVP_Out_P_Min  : REAL;
	EVP_Out_P_Max  : REAL;

	EVP_Out_S_Min  : REAL;
	EVP_Out_S_Max  : REAL;

(*Valve Targets*)
	EVP_In_P_Eng : REAL;
	EVP_In_P_PP  : REAL;

	EVP_In_S_Eng : REAL;
	EVP_In_S_PP  : REAL;

	EVP_Out_P_Eng : REAL;
	EVP_Out_P_PP  : REAL;

	EVP_Out_S_Eng : REAL;
	EVP_Out_S_PP  : REAL;

(*Valve Gains*)
	EVP_In_EVP_K  : REAL;
	EVP_Out_EVP_K : REAL;

	EVP_In_LS_K  : REAL;
	EVP_Out_LS_K : REAL;

(*Valve Softstart*)
	EVP_In_Inc  : REAL;
	EVP_Out_Inc : REAL;

	EVP_In_Dec  : REAL;
	EVP_Out_Dec : REAL;

	LP : BYTE;

	Cycle    : REAL; (*Seconds*)
	TimeMax  : REAL; (*Seconds*)

END_STRUCT
END_TYPE

(* Data type *)
TYPE ST_CAN_NODESTATE :
STRUCT
	Desc : STRING;

	(*Alarm*)
	Alarm  : ST_ALARM;

END_STRUCT
END_TYPE

(* Data type *)
TYPE ST_DE_CYLINDER_POS_CFG :
STRUCT
	TgtLS_In  : REAL;
	TgtLS_Out : REAL;
	TgtLS_Mid : REAL;
	TgtLS_DB  : REAL;

	LS_Limit_In  : BOOL;
	LS_Limit_Out : BOOL;

	Cycle   : REAL; (*Seconds*)
	TimeMax : REAL; (*Seconds*)

	HP : BYTE;
END_STRUCT
END_TYPE

(* Data type *)
TYPE ST_ENGINE_CFG :
STRUCT

	(*Parameters*)
	MaxInc_RPM : REAL; (*RPM/sec*)
	MaxDec_RPM : REAL; (*RPM/sec*)
	DlyDec_sec : REAL;

	Boost_RPM : REAL;
	Max_RPM   : REAL;
	Min_RPM   : REAL;
	Stop_RPM  : REAL;

	HP_Nx_RPM : REAL;
	HP_SF_RPM : REAL;

	LP_CK_RPM : REAL;
	LP_1x_RPM : REAL;
	LP_2x_RPM : REAL;
	LP_3x_RPM : REAL;
	LP_Nx_RPM : REAL;

	N_Winch_WOP : INT;
	N_Winch_WK  : INT;
	N_Winch_WP  : INT;

	Max_Torque : REAL;
	Min_Torque : REAL;

	Inc_RMP_Perc_WOP : REAL;
	Dec_Flow_Perc_WP : REAL;

	Max_HeatExch_P : REAL;

	Cycle : REAL; (*Seconds*)

	EnForceRPM : BOOL;
	EnForceTHR : BOOL;



	(*Coefficients*)
	CycleMaxInc_RPM : REAL;
	CycleMaxDec_RPM : REAL;

	Boost_K : REAL;
	OffDelay_cycl : UINT;

	Inc_RMP_Perc_WOP_K : REAL;
	Dec_Flow_Perc_WP_K : REAL;

END_STRUCT
END_TYPE

(* Data type *)
TYPE ST_KEEL_CFG :
STRUCT
(*Targets*)
	TgtLS_In  : REAL;
	TgtLS_Mid : REAL;
	TgtLS_Out : REAL;

	TgtLS_Safe_In  : REAL;
	TgtLS_Safe_Out : REAL;

	TgtLS_Tack_Off : REAL;

	LS_DB : REAL;

(*Board Limits*)
	Board_P_Min_Out : REAL;
	Board_S_Min_Out : REAL;

(*Valve Limits*)
	EVP_In_SE_Min : REAL; (*mA*)
	EVP_In_SE_Max : REAL;
	EVP_In_SE_Man : REAL;

	EVP_In_FE_Min : REAL;
	EVP_In_FE_Max : REAL;
	EVP_In_FE_Man : REAL;

	EVP_In_Eng_Min : REAL;
	EVP_In_Eng_Max : REAL;
	EVP_In_Eng_Man : REAL;

	EVP_In_P_Empty : REAL; (*bar*)

	EVP_Out_SE_Min : REAL; (*mA*)
	EVP_Out_SE_Max : REAL;
	EVP_Out_SE_Man : REAL;
	EVP_Out_SE_Empty : REAL;

	EVP_Out_FE_Min : REAL;
	EVP_Out_FE_Max : REAL;
	EVP_Out_FE_Man : REAL;

	EVP_Out_Eng_Min : REAL;
	EVP_Out_Eng_Max : REAL;
	EVP_Out_Eng_Man : REAL;

	EVP_Out_Fill_Min  : REAL; (*%*)
	EVP_Out_Fill_Max  : REAL;

	EVP_Out_P_Fill : REAL; (*bar*)

(*Valve Softstart*)
	EVP_In_SE_Inc : REAL;
	EVP_In_SE_Dec : REAL;

	EVP_In_FE_Inc : REAL;
	EVP_In_FE_Dec : REAL;

	EVP_Out_SE_Inc : REAL;
	EVP_Out_SE_Dec : REAL;

	EVP_Out_FE_Inc : REAL;
	EVP_Out_FE_Dec : REAL;

	EVP_In_Eng_Inc : REAL;
	EVP_In_Eng_Dec : REAL;

	EVP_Out_Eng_Inc : REAL;
	EVP_Out_Eng_Dec : REAL;

(*Auto Ease limit*)
	MinLoadSide_Bar   : REAL;
	MaxUnloadSide_Bar : REAL;

(*Valve Gains*)
	EVP_In_Eng_K  : REAL;
	EVP_Out_Eng_K : REAL;

	LP : BYTE;

	Cycle    : REAL; (*Seconds*)
	TimeMax  : REAL; (*Seconds*)

(*Calculated*)
	EVP_Out_Fill_K   : REAL; (*Calculated vs EVP_Out_Eng_Min/Max*)
	EVP_Out_Fill_Off : REAL;



END_STRUCT
END_TYPE

(* Data type *)
TYPE ST_LIFT_KEEL_CFG :
STRUCT
	PMax_Up : REAL; (*Alarm only*)
	PMax_Dw : REAL; (*Alarm only*)

	P500_Up : REAL; (*Usually 15% more than PMax*)
	P500_Dw : REAL; (*Usually 15% more than PMax*)

	P144_F  : REAL; (*Release Max Press.*)
	P144_S  : REAL; (*Release Max Press.*)

	TgtP_Dw   : REAL;
	TgtLS_Up  : REAL;
	TgtLS_SUp : REAL;
	TgtLS_Dw  : REAL;

	P_DB	 : REAL;
	LS_DB    : REAL;
	LS_Dist  : REAL;

	Cycle    : REAL; (*Seconds*)
	TimeMax  : REAL; (*Seconds*)
	Delay_Dw : REAL;

	PP1 : BOOL;
	PP2 : BOOL;
	HP1 : BOOL;
	HP2 : BOOL;
	HP3 : BOOL;
END_STRUCT
END_TYPE

(* Data type *)
TYPE ST_LIFT_PROP_CFG :
STRUCT
	TgtP_Up  : REAL;
	TgtP_Dw  : REAL;
	TgtLS_Up : REAL;
	TgtLS_Dw : REAL;

	P_DB	 : REAL;
	LS_DB    : REAL;

	Cycle    : REAL; (*Seconds*)
	TimeMax  : REAL; (*Seconds*)
	Delay_Up : REAL;
	Delay_Dw : REAL;

	HP_Up : BYTE;
	HP_Dw : BYTE;

END_STRUCT
END_TYPE

(* Data type *)
TYPE ST_LINEAR_CAL :
STRUCT
	K   : REAL;
	Off : REAL;
END_STRUCT
END_TYPE

(* Data type *)
TYPE ST_LOAD_CAL :
STRUCT
	K : REAL;
	C : REAL;
END_STRUCT
END_TYPE

(* Data type *)
TYPE ST_LP_FUNC_CFG :
STRUCT
	SpdA_Min : REAL;
	SpdA_Max : REAL;
	SpdB_Min : REAL;
	SpdB_Max : REAL;

	Spd_Inc : REAL;
	Spd_Dec : REAL;

	A_Spd1 : BOOL;

	SF1_Limit : BOOL;
	SF2_Limit : BOOL;

	Cycle   : REAL; (*Seconds*)
	TimeMax : REAL; (*Seconds*)

(*	PP : BYTE;*)
END_STRUCT
END_TYPE

(* Data type *)
TYPE ST_MAGIC_DOUBLE_CFG :
STRUCT
	P4Max : REAL; (*Alarm only*)
	P2Max : REAL; (*Alarm only*)

	EVPA4  : INT;
	EVPA2  : INT;
	EVPB4  : INT;
	EVPB2  : INT;
	EVPFA4 : INT;
	EVPFA2 : INT;
	EVPFB4 : INT;
	EVPFB2 : INT;

	EVPRA2 : INT;
	EVPRAD : INT;

	TgtLS4_Out : REAL;
	TgtLS4_In  : REAL;
	TgtLS2_Out : REAL;
	TgtLS2_In  : REAL;

	P_DB     : REAL;
	LS_DB    : REAL;

	Cycle    : REAL; (*Seconds*)
	TimeMax  : REAL; (*Seconds*)
	OutDelay : REAL; (*Seconds Pumping 2 & 4*)
	EVTDelay : REAL; (*Seconds before EVT*)

	PP1 : BOOL;
	PP2 : BOOL;
END_STRUCT
END_TYPE

(* Data type *)
TYPE ST_MAST_SETUP :
STRUCT
	Cycle : REAL; (*Seconds*)

	aFSY  : ARRAY[1..4,1..6] OF REAL;
	aBDef : ARRAY[1..4,1..6] OF REAL;
	aTDef : ARRAY[1..4,1..6] OF REAL;


END_STRUCT
END_TYPE

(* Data type *)
TYPE ST_POWERPACK_CFG :
STRUCT
	Hyst_HP : REAL;
	Hyst_LP : REAL;
	Hyst_TM : REAL;	(*Seconds*)

	Thr_HP : REAL;
	Thr_LP : REAL;

	Cycle : REAL;	(*Second*)
END_STRUCT
END_TYPE

(* Data type *)
TYPE ST_PROPULSION_CFG :
STRUCT

	(*Parameters*)
	IdleDB_V  : REAL;
	PropRPM_K : REAL;

	Delay_Off : REAL; (*Second*)
	Cycle     : REAL;

	aThrt_V  : ARRAY [0..10] OF REAL;
	aEng_RPM : ARRAY [0..10] OF REAL;
	aEVP_mA  : ARRAY [0..10] OF REAL;

	(*Coefficients*)
	aEng_K   : ARRAY [0..9] OF REAL;
	aEng_Off : ARRAY [0..9] OF REAL;

	aEVP_K   : ARRAY [0..9] OF REAL;
	aEVP_Off : ARRAY [0..9] OF REAL;


END_STRUCT
END_TYPE

(* Data type *)
TYPE ST_PSX_VALVE_IN :
STRUCT
	Status : UINT;
	Actual : INT;
	Error  : UINT;

END_STRUCT
END_TYPE

(* Data type *)
TYPE ST_PSX_VALVE_OUT :
STRUCT
	Control  : UINT;
	SetPoint : INT;

END_STRUCT
END_TYPE

(* Data type *)
TYPE ST_SE_CYLINDER_CFG :
STRUCT
	Ease    : REAL; (*Usually 15% more than PMax*)
	Cycle   : REAL; (*Seconds*)
	TimeEase: REAL; (*Seconds*)
	TimeMax : REAL; (*Seconds*)
	HP      : BYTE; (*Num. Pumps*)
END_STRUCT
END_TYPE

(* Data type *)
TYPE ST_SE_CYLINDER_POS_CFG :
STRUCT
	Ease : REAL;

	TgtLS_In  : REAL;
	TgtLS_Out : REAL;
	TgtLS_Slow  : REAL;

	LS_Limit_In  : BOOL;
	LS_Limit_Out : BOOL;

	Cycle   : REAL; (*Seconds*)
	TimeEase: REAL; (*Seconds*)
	TimeMax : REAL; (*Seconds*)

	HP : BYTE;

END_STRUCT
END_TYPE

(* Data type *)
TYPE ST_SENSOR_BAR :
STRUCT
	Name : STRING;
	Desc : STRING;

	Raw : REAL;
	Err : BOOL;
	Bar : REAL;

	(*Calib*)
	Cal_K   : REAL;
	Cal_Off : REAL;
	Raw_Off : REAL := 4.0;

	(*Avg*)
	Avg_Buf : ARRAY[0..4] OF REAL;
	Avg_Sum : LREAL;
	Avg_Pos : INT;

	(*Alarm*)
	Alarm : ST_ALARM;

	MinRaw : REAL :=  2.0;
	MaxRaw : REAL := 22.0;
	MinBar : REAL :=  0.0;
	MaxBar : REAL :=  0.0;

	AlErr : BOOL;
	AlMax : BOOL;
	AlMin : BOOL;

	AdverVal : REAL;

END_STRUCT
END_TYPE

(* Data type *)
TYPE ST_SENSOR_KG :
STRUCT
	Name : STRING;

	Raw : REAL;
	Kg  : REAL;

	(*Calib*)
	Cal_K : REAL;
	Cal_C : REAL;

END_STRUCT
END_TYPE

(* Data type *)
TYPE ST_SENSOR_POS :
STRUCT
	Name : STRING;
	Desc : STRING;

	Raw : REAL;
	Err : BOOL;
	Pos : REAL;

	(*Calib*)
	Cal_K   : REAL;
	Cal_Off : REAL;
	Cal_Min : REAL;
	Cal_Max : REAL;
	Cal_Apply : BOOL;

	(*Avg*)
	Avg_Buf : ARRAY[0..4] OF REAL;
	Avg_Sum : LREAL;
	Avg_Pos : INT;

	(*Alarm*)
	Alarm  : ST_ALARM;

	MinRaw : REAL :=  2.0;
	MaxRaw : REAL := 22.0;

END_STRUCT
END_TYPE

(* Data type *)
TYPE ST_SENSOR_SWITCH :
STRUCT
	Name : STRING;
	Desc : STRING;

	(*Alarm*)
	Alarm : ST_ALARM;

	Count  : REAL;


END_STRUCT
END_TYPE

(* Data type *)
TYPE ST_SENSOR_TEMP :
STRUCT
	Name : STRING;
	Desc : STRING;

	Raw : REAL;
	Err : BOOL;
	Deg : REAL;

	(*Calib*)
	Cal_K   : REAL;
	Cal_Off : REAL;

	(*Avg*)
	Avg_Buf : ARRAY[0..4] OF REAL;
	Avg_Sum : LREAL;
	Avg_Pos : INT;

	(*Alarm*)
	Alarm : ST_ALARM;

	MinRaw : REAL :=  2.0;
	MaxRaw : REAL := 22.0;

	LowDeg : REAL;
	HigDeg : REAL;
	MaxDeg : REAL;

	Delay  : REAL;
	Count  : REAL;

	AlErr : BOOL;
	AlLow : BOOL;
	AlHig : BOOL;
	AlMax : BOOL;

	AdverLv  : UINT;
	AdverVal : REAL;

END_STRUCT
END_TYPE

(* Data type *)
TYPE ST_Serial64ByteIn :
STRUCT
	wStatus:WORD;
	aData  :ARRAY[0..63] OF BYTE;
END_STRUCT
END_TYPE

(* Data type *)
TYPE ST_Serial64ByteOut :
STRUCT
	wControl:WORD;
	aData   :ARRAY[0..63] OF BYTE;
END_STRUCT
END_TYPE

(* Data type *)
TYPE ST_TACK_VALVE_CFG :
STRUCT
	Cycle   : REAL; (*Seconds*)
	TimeMax : REAL; (*Seconds*)

	Hyst_HeelH : REAL;
	Hyst_HeelL : REAL;
	Hyst_Time  : REAL;	(*Seconds*)

END_STRUCT
END_TYPE

(* Data type *)
TYPE ST_TRAVELLER_CFG :
STRUCT
	MaxEVPA : REAL;
	MinEVPA : REAL;
	MaxEVPB : REAL;
	MinEVPB : REAL;

	Spd_Inc : REAL;
	Spd_Dec : REAL;

	TgtLS_Min  : REAL;
	TgtLS_Zero : REAL;
	TgtLS_Max  : REAL;

	TgtLS_Tack_Off : REAL;

	LS_DB    : REAL;
	LS_Dist  : REAL;

	LS_Limit : BOOL;

	Cycle    : REAL; (*Seconds*)
	TimeMax  : REAL; (*Seconds*)

	Hyst_HP : REAL;
	Hyst_LP : REAL;
	Hyst_TM : REAL;	(*Seconds*)

	HP      : BYTE; (*Num. Pumps*)
	LP      : BYTE;
END_STRUCT
END_TYPE

(* Data type *)
TYPE ST_VALVE_BAR :
STRUCT
	Name : STRING;

	Bar : REAL;
	mA  : UINT;

	(*Calib*)
	Cal_K   : REAL;
	Cal_Off : REAL;

END_STRUCT
END_TYPE

(* Data type *)
TYPE ST_WB_CFG :
STRUCT
	Cycle   : REAL; (*Seconds*)
	TimeMax_Idle    : REAL;
	TimeMax_Init    : REAL;
	TimeMax_DumpAft : REAL; (*Seconds*)
	TimeMax_DumpFwd : REAL; (*Seconds*)
	TimeMax_MoveAft : REAL; (*Seconds*)
	TimeMax_MoveFwd : REAL; (*Seconds*)

	(*Pump*)
	EVP_Pump_Min : REAL;
	EVP_Pump_Max : REAL;

	EVP_Pump_Inc : REAL;
	EVP_Pump_Dec : REAL;

	EnScoopAF : BOOL;

	LP      : BYTE; (*Num. Pumps*)
END_STRUCT
END_TYPE

(* Data type *)
TYPE ST_WB_VALVE_CFG :
STRUCT
	Cycle   : REAL; (*Seconds*)
	TimeMax : REAL; (*Seconds*)
	PushTime: REAL; (*Seconds*)
	PushP   : REAL; (*Bar*)

	HP      : BYTE; (*Num. Pumps*)
END_STRUCT
END_TYPE

(* Data type *)
TYPE ST_WB_VALVE_LS_CFG :
STRUCT
	Cycle   : REAL; (*Seconds*)
	TimeMax : REAL; (*Seconds*)
	PushTime: REAL; (*Seconds*)
	PushP   : REAL; (*Bar*)

	TgtLS_Half : REAL;
	LS_DB   : REAL;

	HP      : BYTE; (*Num. Pumps*)
END_STRUCT
END_TYPE

(* Data type *)
TYPE ST_WINCHE_CFG :
STRUCT
	Spd1 : ARRAY[1..7] OF REAL;
	Spd2 : ARRAY[1..7] OF REAL;
	Spd3 : ARRAY[1..7] OF REAL;

	A_Spd1 : BOOL;

	P1_Max : REAL;
	P2_Max : REAL;
	P3_Max : REAL;

	Cycle   : REAL; (*Seconds*)
	TimeMax : REAL; (*Seconds*)

(*	PP : BYTE;*)
END_STRUCT
END_TYPE

(* Data type *)
TYPE ST_WINCHE_RAMP_CFG :
STRUCT
	Spd_Min : REAL;
	Spd_Inc : REAL;
	Spd_Dec : REAL;
END_STRUCT
END_TYPE

(* Data type *)
TYPE TxQueue_10 :
STRUCT
	TxCounter      : UINT;
	RxCounter      : UINT;
	NoOfTxMessages : UINT;
	TxMessages     : ARRAY [0..9] OF ARRAY[0..13] OF BYTE;
END_STRUCT
END_TYPE

(* Data type *)
TYPE VARTYPE_EXTCANQUEUE
STRUCT
	dummy : UINT;
	length: UINT;
	cobId : DWORD;
	rxData: ARRAY [0..7] OF USINT;
END_STRUCT
END_TYPE

(* POU MAIN, ST *)
PROGRAM MAIN
VAR CONSTANT
	Cycle_Time : REAL := 0.02; (*20ms*)
END_VAR
VAR
	(*UPS Function to Sstore Persistent Vars*)
	(*fbUPS: FB_S_UPS_CX9020_U900;*)

	(*Cylinders*)
	fbSE301 : FB_SE_CYLINDER_POS;	(* 1*)
	fbSE303 : FB_SE_CYLINDER_POS;	(* 2*)
	fbSE305 : FB_SE_CYLINDER_POS;	(* 3*)
	fbSE307 : FB_SE_CYLINDER_POS;	(* 4*)
	fbSE309 : FB_SE_CYLINDER_POS;	(* 5*)
	fbSE311 : FB_SE_CYLINDER_POS;	(* 6*)

	fbSE501 : FB_DE_CYLINDER;		(* 7*)
	fbSE503 : FB_SE_CYLINDER;		(* 8*)
	fbSE505 : FB_SE_CYLINDER_QR;	(* 9*)

	fbDE601 : FB_LIFTING_PROPELLER;	(*10*)
	fbDE605 : FB_DE_CYLINDER_POS;	(*11*)

	fbSE701 : FB_SE_CYLINDER;		(*12*)
	fbSE703 : FB_SE_CYLINDER;		(*13*)
	fbSE705 : FB_SE_CYLINDER;		(*14*)
	fbSE707 : FB_SE_CYLINDER_POS;	(*15*)
	fbSE709 : FB_SE_CYLINDER_POS;	(*16*)

	fbBSY   : FB_BACKSTAY;			(*17*)
(*	fbSE901 : FB_SE_CYLINDER_POS_FINE;	(*17*) (* Añadir tack y Fine, mejor hacer un unico FB FB_SE_FINE_CYLINDER_POS*)
	fbSE903 : FB_SE_CYLINDER_POS_FINE;	(*18*) (* Con 4 inputs para in Out 2 de ellos fine, y 2 inputs para el tack*)*)

	fbWB   : FB_WATERBALLAST;		(*19*)
	fbWB_A : FB_WB_VALVE;
	fbWB_B : FB_WB_VALVE_LS;
	fbWB_C : FB_WB_VALVE_LS;
	fbWB_D : FB_WB_VALVE;
	fbWB_E : FB_WB_VALVE;
	fbWB_F : FB_WB_VALVE;
	fbWB_G : FB_WB_VALVE;
	fbWB_H : FB_WB_VALVE;
	fbWB_I : FB_WB_VALVE_LS;
	fbWB_J : FB_WB_VALVE;
	fbWB_K : FB_WB_VALVE;
	fbWB_L : FB_WB_VALVE;
	fbWB_M : FB_WB_VALVE;
	fbWB_N : FB_WB_VALVE_LS;
	fbWB_R : FB_WB_VALVE_LS;
	fbWB_S : FB_WB_VALVE_LS;

	fbWB_PUD : FB_WB_VALVE_LS;
    fbWB_PAF : FB_WB_VALVE_LS;
	fbWB_SUD : FB_WB_VALVE_LS;
    fbWB_SAF : FB_WB_VALVE_LS;

	WB_Scoop_Link : BOOL;

	(*Winches*)
	fbW1202	: FB_WINCHE_V2;	(*4*)
	fbW1204	: FB_WINCHE_V2;	(*5*)
	fbW1206	: FB_WINCHE_V2; (*6*)
	fbW1208	: FB_WINCHE_V2;	(*7*)
	fbW1210	: FB_WINCHE_V2;	(*8*)
	fbW1212	: FB_WINCHE_V2;	(*9*)
	fbW1214	: FB_WINCHE_V2;	(*10*)

	fbBoard      : FB_BOARD;	(*11,12*)
	fbKeel       : FB_KEEL;		(*13,19*)

	fbW1602	: FB_WINCHE_V2;	(*14*)
	fbW1604	: FB_WINCHE_V2;	(*15*)

	fbTraveller : FB_TRAVELLER;		(*16*)

	fbBowThr     : FB_LP_FUNC_SF;	(*17*)
	fbBowThrUpDw : FB_LP_FUNC_SF;	(*18*)

	(*Extra functions*)
	fbTackValve : FB_TACK_VALVE;

	fbMastSetup : FB_MAST_SETUP;

	(*SYSTEM STATUS*)
	HMI_Enable : BOOL;
	HMI_ShutDw : BOOL;

	SIEnable : ARRAY[1..3] OF FB_SMART_INPUT;
	SIShutDw : ARRAY[1..3] OF FB_SMART_INPUT;

	SITankEnable   : FB_SMART_INPUT;
	SIEngineEnable : FB_SMART_INPUT;
	SIPropEnable   : FB_SMART_INPUT;
	SIPropUDEnable : FB_SMART_INPUT;

	EventEnable : EN_SMART_INPUT_STATE;
	EventShutDw : EN_SMART_INPUT_STATE;

	SysLabel : STRING;
	LoadLAbel: STRING;
	SysPass  : STRING;
	SysColor : DWORD;
	SysState : WORD := 0;
	SysDClick : BOOL;
	AutoOffCnt : REAL;

END_VAR
VAR PERSISTENT
	aHP_Enable  AT %Q*: ARRAY[1..32] OF BOOL;
	aLP_Enable  AT %Q*: ARRAY[1..32] OF BOOL;
	aWB_Enable  AT %Q*: ARRAY[1..32] OF BOOL;

	aSys_Enable AT %Q*: ARRAY[1..16] OF BOOL;
	(*
	1 - Tank
	2 - SysSail
	3 - SysProp
	4 - EnableHP1
	5 - EnableHP2
	6 - EnablePP1
	7 - EnablePP2
	8 - EngineEnable 
	9 - PropEnable   
	10 - Dimmer_ON
	...
	16 - TackValve
	*)

	Prop_UsedTime 	AT %Q* : REAL;
	W1202_USedTime	AT %Q* : REAL;
	W1204_USedTime	AT %Q* : REAL;
	W1206_USedTime	AT %Q* : REAL;
	W1208_USedTime	AT %Q* : REAL;
	W1210_USedTime	AT %Q* : REAL;
	W1212_USedTime	AT %Q* : REAL;
	W1214_USedTime	AT %Q* : REAL;
	W1602_USedTime	AT %Q* : REAL;
	W1604_USedTime	AT %Q* : REAL;

END_VAR
(*PARAMS;*)
INPUTS;
TANK;

(*SYSTEM STATE: ENABLED / PROP ONLY / DISABLE*)
SIEnable[1](In:= HMI_Enable,  T_Cont:= T#0ms, T_DClk:= T#0ms);
(*SIEnable[2](In:= N103_IN.0 ,  T_Cont:= T#0ms, T_DClk:= T#0ms);
SIEnable[3](In:= N108_IN.1 ,  T_Cont:= T#0ms, T_DClk:= T#0ms);*)
SIShutDw[1](In:= HMI_ShutDw,  T_Cont:= T#1000ms, T_DClk:= T#0ms);
(*SIShutDw[2](In:= N103_IN.1 ,  T_Cont:= T#1000ms, T_DClk:= T#500ms);
SIShutDw[3](In:= N108_IN.0 ,  T_Cont:= T#1000ms, T_DClk:= T#500ms);*)

SITankEnable  (T_Cont:= T#1000ms, T_DClk:=T#0ms);
SIEngineEnable(T_Cont:= T#1000ms, T_DClk:=T#0ms);
SIPropEnable  (T_Cont:= T#1000ms, T_DClk:=T#0ms);
SIPropUDEnable(T_Cont:= T#1000ms, T_DClk:=T#0ms);

IF    SIEnable[1].Event <> NONE THEN EventEnable := SIEnable[1].Event;
ELSIF SIEnable[2].Event <> NONE THEN EventEnable := SIEnable[2].Event;
ELSIF SIEnable[3].Event <> NONE THEN EventEnable := SIEnable[3].Event;
ELSE							     EventEnable := NONE;
END_IF

IF    SIShutDw[1].Event <> NONE THEN EventShutDw := SIShutDw[1].Event;
ELSIF SIShutDw[2].Event <> NONE THEN EventShutDw := SIShutDw[2].Event;
ELSIF SIShutDw[3].Event <> NONE THEN EventShutDw := SIShutDw[3].Event;
ELSE							     EventShutDw := NONE;
END_IF

CASE SysState OF

0:  (*DISABLED*)
	IF EventEnable = INIT_CONTINUOUS (*SysPass = '2005062'*) THEN
		aSys_Enable[2] := TRUE;
		aSys_Enable[3] := TRUE;

		SysState := 2;
	END_IF

	SysLabel := 'SYSTEM$nDISABLED';
	SysColor := 16#000000FF;

1: (*PROP ONLY*)
	IF EventShutDw = INIT_CONTINUOUS THEN
		aSys_Enable[2] := FALSE;
		aSys_Enable[3] := FALSE;
		SysState       := 0;

	ELSIF EventEnable = INIT_CONTINUOUS (*SysPass = '2005062'*) THEN
		aSys_Enable[2] := TRUE;
		aSys_Enable[3] := TRUE;
		SysState       := 2;

	END_IF

	SysLabel := 'ONLY$nPROPULSION';
	SysColor := 16#00000000;

2: (*ENABLE*)
	IF EventShutDw = INIT_CONTINUOUS OR AutoOffCnt > 2400 THEN
		aSys_Enable[2] := FALSE;
		aSys_Enable[3] := TRUE;
		SysPass        := '';
		SysState       := 1;
	END_IF

	SysLabel := 'SAILING$nENABLED';
	SysColor := 16#0000FF00;

END_CASE

IF SITankEnable.Event   = INIT_CONTINUOUS THEN aSys_Enable[1] := NOT aSys_Enable[1]; END_IF
IF SIEngineEnable.Event = INIT_CONTINUOUS THEN aSys_Enable[8] := NOT aSys_Enable[8]; END_IF
IF SIPropEnable.Event   = INIT_CONTINUOUS THEN aSys_Enable[9] := NOT aSys_Enable[9]; END_IF
IF SIPropUDEnable.Event = INIT_CONTINUOUS THEN aHP_Enable[10] := NOT aHP_Enable[10]; END_IF

(*Loadind Status*)
IF PARAMS.Loaded THEN
	LoadLabel := '';
ELSE
	LoadLabel := '(Loading...)';
END_IF


(*Cylinders MF03*)
fbSE301(
	Enable := aHP_Enable[1] AND TANK.Enable AND aSys_Enable[2],
	Ready  := ENGINE.Pump_ON,

	IN_CylIn := INPUTS.B301,
	IN_CylOut:= INPUTS.B302,

	P   :=  P301,
	LS  := LS301,
	CFG := PARAMS.stSE301Cfg,

	OUT_CylIn => EV301,
	OUT_CylOut=> EV302
);
fbSE303(
	Enable := aHP_Enable[2] AND TANK.Enable AND aSys_Enable[2],
	Ready  := ENGINE.Pump_ON,

	IN_CylIn := INPUTS.B303,
	IN_CylOut:= INPUTS.B304,

	P   :=  P303,
	LS  := LS303,
	CFG := PARAMS.stSE303Cfg,

	OUT_CylIn => EV303,
	OUT_CylOut=> EV304
);
fbSE305(
	Enable := aHP_Enable[3] AND TANK.Enable AND aSys_Enable[2],
	Ready  := ENGINE.Pump_ON,

	IN_CylIn := INPUTS.B305,
	IN_CylOut:= INPUTS.B306,

	P   :=  P305,
	LS  := LS305,
	CFG := PARAMS.stSE305Cfg,

	OUT_CylIn => EV305,
	OUT_CylOut=> EV306
);
fbSE307(
	Enable := aHP_Enable[4] AND TANK.Enable AND aSys_Enable[2],
	Ready  := ENGINE.Pump_ON,

	IN_CylIn := INPUTS.B307,
	IN_CylOut:= INPUTS.B308,

	P   :=  P307,
	LS  := LS307,
	CFG := PARAMS.stSE307Cfg,

	OUT_CylIn => EV307,
	OUT_CylOut=> EV308
);
fbSE309(
	Enable := aHP_Enable[5] AND TANK.Enable AND aSys_Enable[2],
	Ready  := ENGINE.Pump_ON,

	IN_CylIn := INPUTS.B309,
	IN_CylOut:= INPUTS.B310,

	P   :=  P309,
	LS  := LS309,
	CFG := PARAMS.stSE309Cfg,

	OUT_CylIn => EV309,
	OUT_CylOut=> EV310
);
fbSE311(
	Enable := aHP_Enable[6] AND TANK.Enable AND aSys_Enable[2],
	Ready  := ENGINE.Pump_ON,

	IN_CylIn := INPUTS.B311,
	IN_CylOut:= INPUTS.B312,

	P   :=  P311,
	LS  := LS311,
	CFG := PARAMS.stSE311Cfg,

	OUT_CylIn => EV311,
	OUT_CylOut=> EV312
);

EVP313.Bar := 10000;
IF fbSE301.OUT_CylOut THEN EVP313.Bar := MIN(fbSE301.OUT_Ease, EVP313.Bar); END_IF
IF fbSE303.OUT_CylOut THEN EVP313.Bar := MIN(fbSE303.OUT_Ease, EVP313.Bar); END_IF
IF fbSE305.OUT_CylOut THEN EVP313.Bar := MIN(fbSE305.OUT_Ease, EVP313.Bar); END_IF
IF fbSE307.OUT_CylOut THEN EVP313.Bar := MIN(fbSE307.OUT_Ease, EVP313.Bar); END_IF
IF fbSE309.OUT_CylOut THEN EVP313.Bar := MIN(fbSE309.OUT_Ease, EVP313.Bar); END_IF
IF fbSE311.OUT_CylOut THEN EVP313.Bar := MIN(fbSE311.OUT_Ease, EVP313.Bar); END_IF
IF EVP313.Bar = 10000 THEN EVP313.Bar := 0.0; END_IF

(*Cylinders MF05*)
fbSE501(
	Enable := aHP_Enable[7] AND TANK.Enable AND aSys_Enable[2],
	Ready  := ENGINE.Pump_ON,

	IN_CylIn := INPUTS.B501,
	IN_CylOut:= INPUTS.B502,

	P_In  := P501,
	P_Out := P507,
	CFG   := PARAMS.stSE501Cfg,

	OUT_CylIn => EV501,
	OUT_CylOut=> EV502
);
EV507 := EV502;
EV508 := EV501;

fbSE503(
	Enable := aHP_Enable[8] AND TANK.Enable AND aSys_Enable[2],
	Ready  := ENGINE.Pump_ON,

	IN_CylIn := INPUTS.B503,
	IN_CylOut:= INPUTS.B504,

	P   := P503,
	CFG := PARAMS.stSE503Cfg,

	OUT_CylIn => EV503,
	OUT_CylOut=> EV504
);
fbSE505(
	Enable := aHP_Enable[9] AND TANK.Enable AND aSys_Enable[2],
	Ready  := ENGINE.Pump_ON,

	IN_CylIn := INPUTS.B505,
	IN_CylOut:= INPUTS.B506,
	IN_CylQR := INPUTS.B506Q,

	P   := P505,
	CFG := PARAMS.stSE505Cfg,

	OUT_CylIn => EV505,
	OUT_CylOut=> EV506
);

EVP513.Bar := 10000;
IF fbSE501.OUT_CylOut THEN EVP513.Bar := MIN(fbSE501.OUT_Ease, EVP513.Bar); END_IF
IF fbSE503.OUT_CylOut THEN EVP513.Bar := MIN(fbSE503.OUT_Ease, EVP513.Bar); END_IF
IF fbSE505.OUT_CylOut THEN EVP513.Bar := MIN(fbSE505.OUT_Ease, EVP513.Bar); END_IF
IF EVP513.Bar = 10000 THEN EVP513.Bar := 0.0; END_IF

(*Cylinders MF06*)
fbDE601(
	Enable := aHP_Enable[10] AND TANK.Enable AND aSys_Enable[3],
	ReadyUp:= ENGINE.fbPropulsion.Idle,
	Clear  := ALARMS.Clear,

	IN_CylIn := INPUTS.B603,
	IN_CylOut:= INPUTS.B601,

	P_In  :=  P603,
	P_Out :=  P601,
	LS    := LS601,
	CFG   := PARAMS.stDE601Cfg,

	OUT_EV1=> EV601, (*Pump OUT*)
	OUT_EV2=> EV602, (*Ease OUT*)
	OUT_EV3=> EV603, (*Pump IN*)
	OUT_EV4=> EV604  (*Ease IN*)
);
fbDE605(
	Enable := aHP_Enable[11] AND TANK.Enable AND aSys_Enable[2],
	Ready  := ENGINE.Pump_ON,

	IN_CylIn := INPUTS.B607,
	IN_CylOut:= INPUTS.B605,
	IN_CylMid:=INPUTS.B606,

	P_In  :=  P607,
	P_Out :=  P605,
	LS    := LS605,
	CFG   := PARAMS.stDE605Cfg,

	OUT_EV1 => EV605, (*Pump OUT*)
	OUT_EV2 => EV606, (*Ease OUT*)
	OUT_EV3 => EV607, (*Pump IN*)
	OUT_EV4 => EV608  (*Ease IN*)
);

(*Cylinders MF07*)
fbSE701(
	Enable := aHP_Enable[12] AND TANK.Enable AND aSys_Enable[2],
	Ready  := ENGINE.Pump_ON,

	IN_CylIn := INPUTS.B701,
	IN_CylOut:= INPUTS.B702,

	P   :=  P701,
	CFG := PARAMS.stSE701Cfg,

	OUT_CylIn => EV701,
	OUT_CylOut=> EV702
);
fbSE703(
	Enable := aHP_Enable[13] AND TANK.Enable AND aSys_Enable[2],
	Ready  := ENGINE.Pump_ON,

	IN_CylIn := INPUTS.B703,
	IN_CylOut:= INPUTS.B704,

	P   :=  P703,
	CFG := PARAMS.stSE703Cfg,

	OUT_CylIn => EV703,
	OUT_CylOut=> EV704
);
fbSE705(
	Enable := aHP_Enable[14] AND TANK.Enable AND aSys_Enable[2],
	Ready  := ENGINE.Pump_ON,

	IN_CylIn := INPUTS.B705,
	IN_CylOut:= INPUTS.B706,

	P   :=  P705,
	CFG := PARAMS.stSE705Cfg,

	OUT_CylIn => EV705,
	OUT_CylOut=> EV706
);
fbSE707(
	Enable := aHP_Enable[15] AND TANK.Enable AND aSys_Enable[2],
	Ready  := ENGINE.Pump_ON,

	IN_CylIn := INPUTS.B707,
	IN_CylOut:= INPUTS.B708,

	P   :=  P707,
	LS  := LS707,
	CFG := PARAMS.stSE707Cfg,

	OUT_CylIn => EV707,
	OUT_CylOut=> EV708
);
fbSE709(
	Enable := aHP_Enable[16] AND TANK.Enable AND aSys_Enable[2],
	Ready  := ENGINE.Pump_ON,

	IN_CylIn := INPUTS.B709,
	IN_CylOut:= INPUTS.B710,

	P   :=  P709,
	LS  := LS709,
	CFG := PARAMS.stSE709Cfg,

	OUT_CylIn => EV709,
	OUT_CylOut=> EV710
);

EVP709.Bar := 10000;
IF fbSE701.OUT_CylOut THEN EVP709.Bar := MIN(fbSE701.OUT_Ease, EVP709.Bar); END_IF
IF fbSE703.OUT_CylOut THEN EVP709.Bar := MIN(fbSE703.OUT_Ease, EVP709.Bar); END_IF
IF fbSE705.OUT_CylOut THEN EVP709.Bar := MIN(fbSE705.OUT_Ease, EVP709.Bar); END_IF
IF fbSE707.OUT_CylOut THEN EVP709.Bar := MIN(fbSE707.OUT_Ease, EVP709.Bar); END_IF
IF fbSE709.OUT_CylOut THEN EVP709.Bar := MIN(fbSE709.OUT_Ease, EVP709.Bar); END_IF
IF EVP709.Bar = 10000 THEN EVP709.Bar := 0.0; END_IF

(*Cylinders MF09*)
fbBSY(
	Enable := aHP_Enable[17] AND TANK.Enable AND aSys_Enable[2],
	Ready  := ENGINE.Pump_ON,

	IN_P_In  := INPUTS.B901,
	IN_P_Out := INPUTS.B902,
	IN_S_In  := INPUTS.B903,
	IN_S_Out := INPUTS.B904,

	P_P  :=  P901,
	P_S  :=  P903,
	LS_P := LS901,
	LS_S := LS903,
	CFG  := PARAMS.stSE901Cfg,

	OUT_P_In => EV901,
	OUT_P_Out=> EV902,
	OUT_S_In => EV903,
	OUT_S_Out=> EV904
);
(*fbSE901(
	Enable := aHP_Enable[17] AND TANK.Enable AND aSys_Enable[2],
	Ready  := ENGINE.Pump_ON,

	IN_CylIn := INPUTS.B901,
	IN_CylOut:= INPUTS.B902,

	P   :=  P901,
	LS  := LS901,
	CFG := PARAMS.stSE901Cfg,

	OUT_CylIn => EV901,
	OUT_CylOut=> EV902
);
fbSE903(
	Enable := aHP_Enable[18] AND TANK.Enable AND aSys_Enable[2],
	Ready  := ENGINE.Pump_ON,

	IN_CylIn := INPUTS.B903,
	IN_CylOut:= INPUTS.B904,

	P   :=  P903,
	LS  := LS903,
	CFG := PARAMS.stSE903Cfg,

	OUT_CylIn => EV903,
	OUT_CylOut=> EV904
);*)

(*WATER BALLAST***************************************************************)
fbWB(
	Enable := aHP_Enable[19] AND TANK.Enable AND aSys_Enable[2],
	Ready  := ENGINE.Pump_ON,
	Perc   := POWERPACK.LP_Perc,

	IN_P_Fwd := INPUTS.BWB_P_Fwd,
	IN_P_Aft := INPUTS.BWB_P_Aft,
	IN_S_Fwd := INPUTS.BWB_S_Fwd,
	IN_S_Aft := INPUTS.BWB_S_Aft,
	IN_Fill  := INPUTS.BWB_Fill,
	IN_12    := INPUTS.BWB_12,
	IN_Dump  := INPUTS.BWB_Dump,
	IN_Move  := INPUTS.BWB_Move,
	IN_Stop  := INPUTS.BWB_Stop,

	SF_P_Aft := NOT SF021,
	SF_P_Fwd := NOT SF022,
	SF_S_Aft := NOT SF023,
	SF_S_Fwd := NOT SF024,

	WB_A := fbWB_A,
	WB_B := fbWB_B,
	WB_C := fbWB_C,
	WB_D := fbWB_D,
	WB_E := fbWB_E,
	WB_F := fbWB_F,
	WB_G := fbWB_G,
	WB_H := fbWB_H,
	WB_I := fbWB_I,
	WB_J := fbWB_J,
	WB_K := fbWB_K,
	WB_L := fbWB_L,
	WB_M := fbWB_M,
	WB_N := fbWB_N,
	WB_R := fbWB_R,
	WB_S := fbWB_S,

	WB_PUD := fbWB_PUD,
    WB_PAF := fbWB_PAF,
	WB_SUD := fbWB_SUD,
    WB_SAF := fbWB_SAF,

	CFG:= PARAMS.stWBCfg,

	EVP_Pump => EVP1608_9
);
EVP1608_9 := -EVP1608_9; (*Using B*)

fbWB_G(
	Enable:= aHP_Enable[19] AND TANK.Enable AND aSys_Enable[2],
	Manual:= fbWB.Manual,
	SF_Open := SF1901,
	SF_Close:= SF1903,
	P  := P2500,
	CFG:= PARAMS.stWBValveSFCfg,
	OUT_Open => EV1903,
	OUT_Close=> EV1901,
);
fbWB_PUD(
	Enable:= aHP_Enable[19] AND TANK.Enable AND aSys_Enable[2],
	Manual:= fbWB.Manual,
	R_Open  := fbWB_PAF.IN_Hmi_Open AND WB_Scoop_Link,
	R_Close := fbWB_PAF.IN_Hmi_Close AND WB_Scoop_Link,
	LS := LS1905,
	P  := P2500,
	CFG:= PARAMS.stWBValveLSCfg,
	OUT_Open => EV1907, (*dw*)
	OUT_Close=> EV1905, (*up*)
);
fbWB_H(
	Enable:= aHP_Enable[19] AND TANK.Enable AND aSys_Enable[2],
	Manual:= fbWB.Manual,
	SF_Open := SF1909,
	SF_Close:= SF1911,
	P  := P2500,
	CFG:= PARAMS.stWBValveSFCfg,
	OUT_Open => EV1911,
	OUT_Close=> EV1909,
);

fbWB_C(
	Enable:= aHP_Enable[19] AND TANK.Enable AND aSys_Enable[2],
	Manual:= fbWB.Manual,
	LS := LS2001,
	P  := P2500,
	CFG:= PARAMS.stWBValveLSCfg,
	OUT_Open => EV2001,
	OUT_Close=> EV2003,
);
fbWB_PAF(
	Enable:= aHP_Enable[19] AND TANK.Enable AND aSys_Enable[2],
	Manual:= fbWB.Manual,
	R_Open  := fbWB_PUD.IN_Hmi_Open AND WB_Scoop_Link,
	R_Close := fbWB_PUD.IN_Hmi_Close AND WB_Scoop_Link,
	LS := LS2005,
	P  := P2500,
	CFG:= PARAMS.stWBValveLSCfg,
	OUT_Open => EV2007,
	OUT_Close=> EV2005,
);
fbWB_L(
	Enable:= aHP_Enable[19] AND TANK.Enable AND aSys_Enable[2],
	Manual:= fbWB.Manual,
	SF_Open := SF2009,
	SF_Close:= SF2011,
	P  := P2500,
	CFG:= PARAMS.stWBValveSFCfg,
	OUT_Open => EV2011,
	OUT_Close=> EV2009,
);


fbWB_A(
	Enable:= aHP_Enable[19] AND TANK.Enable AND aSys_Enable[2],
	Manual:= fbWB.Manual,
	SF_Open := SF2101,
	SF_Close:= SF2103,
	P  := P2500,
	CFG:= PARAMS.stWBValveSFCfg,
	OUT_Open => EV2103,
	OUT_Close=> EV2101,
);
fbWB_D(
	Enable:= aHP_Enable[19] AND TANK.Enable AND aSys_Enable[2],
	Manual:= fbWB.Manual,
	SF_Open := SF2105,
	SF_Close:= SF2107,
	P  := P2500,
	CFG:= PARAMS.stWBValveSFCfg,
	OUT_Open => EV2107,
	OUT_Close=> EV2105,
);
fbWB_E(
	Enable:= aHP_Enable[19] AND TANK.Enable AND aSys_Enable[2],
	Manual:= fbWB.Manual,
	SF_Open := SF2109,
	SF_Close:= SF2111,
	P  := P2500,
	CFG:= PARAMS.stWBValveSFCfg,
	OUT_Open => EV2111,
	OUT_Close=> EV2109,
);

fbWB_SUD(
	Enable:= aHP_Enable[19] AND TANK.Enable AND aSys_Enable[2],
	Manual:= fbWB.Manual,
	R_Open  := fbWB_SAF.IN_Hmi_Open AND WB_Scoop_Link,
	R_Close := fbWB_SAF.IN_Hmi_Close AND WB_Scoop_Link,
	LS := LS2201,
	P  := P2500,
	CFG:= PARAMS.stWBValveLSCfg,
	OUT_Open => EV2203,
	OUT_Close=> EV2201,
);
fbWB_M(
	Enable:= aHP_Enable[19] AND TANK.Enable AND aSys_Enable[2],
	Manual:= fbWB.Manual,
	SF_Open := SF2205,
	SF_Close:= SF2207,
	P  := P2500,
	CFG:= PARAMS.stWBValveSFCfg,
	OUT_Open => EV2207,
	OUT_Close=> EV2205,
);
fbWB_K(
	Enable:= aHP_Enable[19] AND TANK.Enable AND aSys_Enable[2],
	Manual:= fbWB.Manual,
	SF_Open := SF2209,
	SF_Close:= SF2211,
	P  := P2500,
	CFG:= PARAMS.stWBValveSFCfg,
	OUT_Open => EV2211,
	OUT_Close=> EV2209,
);

fbWB_S(
	Enable:= aHP_Enable[19] AND TANK.Enable AND aSys_Enable[2],
	Manual:= fbWB.Manual,
	LS := LS2301,
	P  := P2500,
	CFG:= PARAMS.stWBValveLSCfg,
	OUT_Open => EV2301,
	OUT_Close=> EV2303,
);
fbWB_B(
	Enable:= aHP_Enable[19] AND TANK.Enable AND aSys_Enable[2],
	Manual:= fbWB.Manual,
	LS := LS2305,
	P  := P2500,
	CFG:= PARAMS.stWBValveLSCfg,
	OUT_Open => EV2305,
	OUT_Close=> EV2307,
);
fbWB_F(
	Enable:= aHP_Enable[19] AND TANK.Enable AND aSys_Enable[2],
	Manual:= fbWB.Manual,
	SF_Open := SF2309,
	SF_Close:= SF2311,
	P  := P2500,
	CFG:= PARAMS.stWBValveSFCfg,
	OUT_Open => EV2311,
	OUT_Close=> EV2309,
);

fbWB_SAF(
	Enable:= aHP_Enable[19] AND TANK.Enable AND aSys_Enable[2],
	Manual:= fbWB.Manual,
	R_Open  := fbWB_SUD.IN_Hmi_Open AND WB_Scoop_Link,
	R_Close := fbWB_SUD.IN_Hmi_Close AND WB_Scoop_Link,
	LS := LS2401,
	P  := P2500,
	CFG:= PARAMS.stWBValveLSCfg,
	OUT_Open => EV2403,
	OUT_Close=> EV2401,
);
fbWB_J(
	Enable:= aHP_Enable[19] AND TANK.Enable AND aSys_Enable[2],
	Manual:= fbWB.Manual,
	SF_Open := SF2405,
	SF_Close:= SF2407,
	P  := P2500,
	CFG:= PARAMS.stWBValveSFCfg,
	OUT_Open => EV2407,
	OUT_Close=> EV2405,
);
fbWB_R(
	Enable:= aHP_Enable[19] AND TANK.Enable AND aSys_Enable[2],
	Manual:= fbWB.Manual,
	LS := LS2409,
	P  := P2500,
	CFG:= PARAMS.stWBValveLSCfg,
	OUT_Open => EV2409,
	OUT_Close=> EV2411,
);

fbWB_N(
	Enable:= aHP_Enable[19] AND TANK.Enable AND aSys_Enable[2],
	Manual:= fbWB.Manual,
	LS := LS2501,
	P  := P2500,
	CFG:= PARAMS.stWBValveLSCfg,
	OUT_Open => EV2501,
	OUT_Close=> EV2503,
);
EV2502 := EV2503;
EV2504 := EV2501;

fbWB_I(
	Enable:= aHP_Enable[19] AND TANK.Enable AND aSys_Enable[2],
	Manual:= fbWB.Manual,
	LS := LS2505,
	P  := P2500,
	CFG:= PARAMS.stWBValveLSCfg,
	OUT_Open => EV2505,
	OUT_Close=> EV2507,
);
EV2506 := EV2507;
EV2508 := EV2505;

(*WINCHES*********************************************************************)
fbW1202(
	Enable:= aLP_Enable[4] AND TANK.Enable AND ENGINE.Pump_ON AND aSys_Enable[2],
	Ready := POWERPACK.WinchReady,(* AND ENGINE.Pump_ON,*)
	Perc  := POWERPACK.LP_Perc,

	IN_1    := INPUTS.B1202_1,
	IN_2    := INPUTS.B1202_2,
	IN_3    := INPUTS.B1202_G,

	P_A := P1202,
	P_B := P1203,
	CFG := PARAMS.stW1202Cfg,
	RAMP:= PARAMS.stWRampCfg,

	OUT_TWC => EVP1202_3,
);
fbW1204(
	Enable:= aLP_Enable[5] AND TANK.Enable AND ENGINE.Pump_ON AND aSys_Enable[2],
	Ready := POWERPACK.WinchReady,(* AND ENGINE.Pump_ON,*)
	Perc  := POWERPACK.LP_Perc,

	IN_1    := INPUTS.B1204_1,
	IN_2    := INPUTS.B1204_2,
	IN_3    := INPUTS.B1204_G,

	P_A := P1204,
	P_B := P1205,
	CFG := PARAMS.stW1204Cfg,
	RAMP:= PARAMS.stWRampCfg,

	OUT_TWC => EVP1204_5,
);
fbW1206(
	Enable:= aLP_Enable[6] AND TANK.Enable AND ENGINE.Pump_ON AND aSys_Enable[2],
	Ready := POWERPACK.WinchReady,(* AND ENGINE.Pump_ON,*)
	Perc  := POWERPACK.LP_Perc,

	IN_1    := INPUTS.B1206_1,
	IN_2    := INPUTS.B1206_2,
	IN_3    := INPUTS.B1206_G,

	Override := INPUTS.Override_ON,

	P_A := P1206,
	P_B := P1207,
	CFG := PARAMS.stW1206Cfg,
	RAMP:= PARAMS.stWRampCfg,

	OUT_TWC => EVP1206_7,
);
fbW1208(
	Enable:= aLP_Enable[7] AND TANK.Enable AND ENGINE.Pump_ON AND aSys_Enable[2],
	Ready := POWERPACK.WinchReady,(* AND ENGINE.Pump_ON,*)
	Perc  := POWERPACK.LP_Perc,

	IN_1    := INPUTS.B1208_1,
	IN_2    := INPUTS.B1208_2,
	IN_3    := INPUTS.B1208_G,

	P_A := P1208,
	P_B := P1209,
	CFG := PARAMS.stW1208Cfg,
	RAMP:= PARAMS.stWRampCfg,

	OUT_TWC => EVP1208_9,
);
fbW1210(
	Enable:= aLP_Enable[8] AND TANK.Enable AND ENGINE.Pump_ON AND aSys_Enable[2],
	Ready := POWERPACK.WinchReady,(* AND ENGINE.Pump_ON,*)
	Perc  := POWERPACK.LP_Perc,

	IN_1    := INPUTS.B1210_1,
	IN_2    := INPUTS.B1210_2,
	IN_3    := INPUTS.B1210_G,

	P_A := P1210,
	P_B := P1211,
	CFG := PARAMS.stW1210Cfg,
	RAMP:= PARAMS.stWRampCfg,

	OUT_TWC => EVP1210_1,
);
fbW1212(
	Enable:= aLP_Enable[9] AND TANK.Enable AND ENGINE.Pump_ON AND aSys_Enable[2],
	Ready := POWERPACK.WinchReady,(* AND ENGINE.Pump_ON,*)
	Perc  := POWERPACK.LP_Perc,

	IN_1    := INPUTS.B1212_1,
	IN_2    := INPUTS.B1212_2,
	IN_3    := INPUTS.B1212_G,

	P_A := P1212,
	P_B := P1213,
	CFG := PARAMS.stW1212Cfg,
	RAMP:= PARAMS.stWRampCfg,

	OUT_TWC => EVP1212_3,
);
fbW1214(
	Enable:= aLP_Enable[10] AND TANK.Enable AND ENGINE.Pump_ON AND aSys_Enable[2],
	Ready := POWERPACK.WinchReady,(* AND ENGINE.Pump_ON,*)
	Perc  := POWERPACK.LP_Perc,

	IN_1    := INPUTS.B1214_1,
	IN_2    := INPUTS.B1214_2,
	IN_3    := INPUTS.B1214_G,

	P_A := P1214,
	P_B := P1215,
	CFG := PARAMS.stW1214Cfg,
	RAMP:= PARAMS.stWRampCfg,

	OUT_TWC => EVP1214_5,
);

fbBoard(
	Enable := aLP_Enable[11] AND TANK.Enable AND aSys_Enable[2],
	Ready  := ENGINE.Pump_ON,

	EngReady := ENGINE.Engine_ON AND NOT ENGINE.Propulion_ON,
	Latching := aLP_Enable[12],

	Keel_Pos := fbKeel.LS_Pos,
	Keel_Err := fbKeel.LS_Err,

	IN_P := INPUTS.BBoardP,
	IN_S := INPUTS.BBoardS,
	IN_C := INPUTS.BBoardC,

	PA_P := P802,
	PA_S := P804,
	PB_P := P1216,
	PB_S := P1219,

	LS_P := LS801,
	LS_S := LS803,

	SF_P := SF801,
	SF_S := SF803,

	CFG := PARAMS.stBoardCfg,

	OUT_TWC_P => EVP1216_7,
	OUT_TWC_S => EVP1218_9,

	OUT_EVB_P => EV801,
	OUT_EVB_S => EV803,

	OUT_EVT_P => EV802,
	OUT_EVT_S => EV804
);
EVP1218_9 := -EVP1218_9; (*Inverted rev 19*)

fbKeel(
	Enable := aLP_Enable[13] AND TANK.Enable AND aSys_Enable[2] AND (NOT SF1002.Alarm.Alarm OR fbKeel.BypassSF),
	Ready  := ENGINE.Pump_ON,

	EngReady := ENGINE.Engine_ON AND NOT ENGINE.Propulion_ON,
	Latching := aLP_Enable[19],

	AutoEase := aLP_Enable[20],

	IN_I := INPUTS.BKeelS,
	IN_O := INPUTS.BKeelP,
	IN_C := INPUTS.BKeelC,
	IN_F := INPUTS.BKeelF,
	IN_T := INPUTS.BKeelT,

	LS_BOARD_P := LS801,
	LS_BOARD_S := LS803,

	P_I :=  P1001,
	P_O :=  P1002,
	LS1 := LS1001,
	LS2 := LS1002,

	CFG := PARAMS.stKeelCfg,

	EV_Eng_PI => EV1001,
	EV_Eng_EI => EV1003,
	EV_Eng_PO => EV1002,
	EV_Eng_EO => EV1004,
	EV_PP_I  => EV1012,
	EV_PP_O  => EV1011,

(*	EVP_Eng_I : UINT;*)
(*	EVP_Eng_O : UINT;*)

	EVP_SE_I  => EVP1006,
	EVP_SE_O  => EVP1007,
	EVP_FE_I  => EVP1008,
	EVP_FE_O  => EVP1009,

	P_Fill  => EVP1005.Bar,
	P_Empty => EVP1010.Bar,

	EVP_Fill => EVP1220_1,

);


fbW1602(
	Enable:= aLP_Enable[14] AND TANK.Enable AND ENGINE.Pump_ON AND aSys_Enable[2],
	Ready := POWERPACK.WinchReady,(* AND ENGINE.Pump_ON,*)
	Perc  := POWERPACK.LP_Perc,

	IN_1    := INPUTS.B1602_1,
	IN_2    := INPUTS.B1602_2,
	IN_3    := INPUTS.B1602_G,

	P_A := P1602,
	P_B := P1603,
	CFG := PARAMS.stW1602Cfg,
	RAMP:= PARAMS.stWRampCfg,

	OUT_TWC => EVP1602_3,
);
fbW1604(
	Enable:= aLP_Enable[15] AND TANK.Enable AND ENGINE.Pump_ON AND aSys_Enable[2],
	Ready := POWERPACK.WinchReady,(* AND ENGINE.Pump_ON,*)
	Perc  := POWERPACK.LP_Perc,

	IN_1    := INPUTS.B1604_1,
	IN_2    := INPUTS.B1604_2,
	IN_3    := INPUTS.B1604_G,

	P_A := P1604,
	P_B := P1605,
	CFG := PARAMS.stW1604Cfg,
	RAMP:= PARAMS.stWRampCfg,

	OUT_TWC => EVP1604_5,
);

fbTraveller(
	Enable := aLP_Enable[16] AND TANK.Enable AND aSys_Enable[2],
	Ready  := ENGINE.Pump_ON,
	Perc   := POWERPACK.LP_Perc,

	IN_A := INPUTS.BTravA,
	IN_B := INPUTS.BTravB,
	IN_T := INPUTS.BTravT,
	IN_D := INPUTS.BTravD,

	P_A :=  P1301,
	P_B :=  P1302,
	LS  := LS1303,
	CFG := PARAMS.stTravellerCfg,

	OUT_EVRA => EV1301,
	OUT_EVRB => EV1302,
	OUT_EVAB => EV1303,
	OUT_TWC  => EVP1606_7
);
EV905 := EV908 := fbTraveller.OUT_EVPA;
EV907 := EV906 := fbTraveller.OUT_EVPB;

fbBowThr(
	Enable:= aLP_Enable[17] AND TANK.Enable AND ENGINE.Pump_ON AND aSys_Enable[2],
	Ready := POWERPACK.WinchReady AND ENGINE.Pump_ON AND (SF404 OR NOT PARAMS.stBowThrUpDwCfg.SF2_Limit),
	Perc  := POWERPACK.LP_Perc,

	IN_1 := INPUTS.BBowThrP,
	IN_2 := INPUTS.BBowThrS,

	CFG := PARAMS.stBowThrCfg,

	OUT_TWC => EVP402_3,
);
fbBowThrUpDw(
	Enable:= aLP_Enable[18] AND TANK.Enable AND ENGINE.Pump_ON AND aSys_Enable[2],
	Ready := POWERPACK.WinchReady AND ENGINE.Pump_ON,
	Perc  := POWERPACK.LP_Perc,

	IN_1 := INPUTS.BBowThrU,
	IN_2 := INPUTS.BBowThrD,

	IN_SF1 := SF405,
	IN_SF2 := SF404,

	CFG := PARAMS.stBowThrUpDwCfg,

	OUT_TWC => EVP404_5,
);

fbTackValve(
	Enable := aSys_Enable[16] AND NOT SF000.Alarm.Alarm (*AND aSys_Enable[2]*),
	Clear  := ALARMS.Clear,

	Heel_Ready  := TOFARO.Recv_Live,
	Heel_Value  := TOFARO.rHeel,

	Port_Ready := N21_DI0_CH7_4,
	Port_Open  := N22_DI0_CH7_4,
	Port_Close := N22_DI1_CH7_2,

	Stbd_Ready := N21_DI1_CH7_2,
	Stbd_Open  := N22_DI6_CH8_4,
	Stbd_Close := N22_DI7_CH8_2,

	CFG := PARAMS.stTackValveCfg,

	OUT_Port_Open  => N36_DO5_CH4_2,
	OUT_Port_Close => N36_DO4_CH4_4,
	OUT_Stbd_Open  => N36_DO1_CH2_2,
	OUT_Stbd_Close => N36_DO0_CH2_4,

);

fbMastSetup(
	IN_MS  := N116_IN.0,
	IN_1th := N109_IN.2,
	IN_2th := N109_IN.4,
	IN_3th := N109_IN.3,
	IN_FH  := N109_IN.0,

	IN_HS := N117_IN.1,
	IN_A3 := N108_IN.0,
	IN_F0 := N108_IN.4,
	IN_J2 := N108_IN.2,
	IN_J4 := N108_IN.3,

	END_MS := N109_IN.5 OR N109_IN.6 OR N109_IN.7,
	END_HS := N108_IN.5 OR N108_IN.6 OR N108_IN.7,

	FSY_P   :=  P309,
	FSY_LS  := LS309,

	BDef_P  :=  P707,
	BDef_LS := LS707,

	TDef_P  :=  P709,
	TDef_LS := LS709,

	TABLE := PARAMS.stMastSetup,

	FSY_In  => fbSE309.IN_RemIn,
	FSY_Out => fbSE309.IN_RemOut,

	BDef_In  => fbSE707.IN_RemIn,
	BDef_Out => fbSE707.IN_RemOut,

	TDef_In  => fbSE709.IN_RemIn,
	TDef_Out => fbSE709.IN_RemOut
);

(*Cylinders*)
IF fbSE301.State <> 0
OR fbSE303.State <> 0
OR fbSE305.State <> 0
OR fbSE307.State <> 0
OR fbSE309.State <> 0
OR fbSE311.State <> 0

OR fbSE501.State <> 0
OR fbSE503.State <> 0
OR fbSE505.State <> 0

OR fbDE601.State <> 0
OR fbDE605.State <> 0

OR fbSE701.State <> 0
OR fbSE703.State <> 0
OR fbSE705.State <> 0
OR fbSE707.State <> 0
OR fbSE709.State <> 0

OR fbBSY.State_P <> 0
OR fbBSY.State_S <> 0
(*
OR fbSE901.State <> 0
OR fbSE903.State <> 0
*)
(*Water Ballast*)
OR fbWB.State <> 0
OR fbWB_A.State <> 0
OR fbWB_B.State <> 0
OR fbWB_C.State <> 0
OR fbWB_D.State <> 0
OR fbWB_E.State <> 0
OR fbWB_F.State <> 0
OR fbWB_G.State <> 0
OR fbWB_H.State <> 0
OR fbWB_I.State <> 0
OR fbWB_J.State <> 0
OR fbWB_K.State <> 0
OR fbWB_L.State <> 0
OR fbWB_M.State <> 0
OR fbWB_N.State <> 0
OR fbWB_R.State <> 0
OR fbWB_S.State <> 0
OR fbWB_PUD.State <> 0
OR fbWB_PAF.State <> 0
OR fbWB_SUD.State <> 0
OR fbWB_SAF.State <> 0

(*Winches*)
OR fbW1202.State <> 0
OR fbW1204.State <> 0
OR fbW1206.State <> 0
OR fbW1208.State <> 0
OR fbW1210.State <> 0
OR fbW1212.State <> 0
OR fbW1214.State <> 0

OR fbW1602.State <> 0
OR fbW1604.State <> 0

OR fbBoard.State       <> 0
OR fbKeel.State        <> 0
OR fbTraveller.State   <> 0

OR fbBowThr.State     <> 0
OR fbBowThrUpDw.State <> 0

OR NOT aSys_Enable[2]
THEN AutoOffCnt := 0.0;
ELSE AutoOffCnt := AutoOffCnt + Cycle_Time;
END_IF

POWERPACK;
ENGINE;
ALARMS;
OUTPUTS;
TOFARO;

IF ENGINE.fbPropulsion.MoveEV THEN Prop_UsedTime := Prop_UsedTime + Cycle_Time; END_IF

IF fbW1202.OUT_TWC <> 0 THEN W1202_USedTime := W1202_USedTime + Cycle_Time; END_IF
IF fbW1204.OUT_TWC <> 0 THEN W1202_USedTime := W1202_USedTime + Cycle_Time; END_IF
IF fbW1206.OUT_TWC <> 0 THEN W1202_USedTime := W1202_USedTime + Cycle_Time; END_IF
IF fbW1208.OUT_TWC <> 0 THEN W1202_USedTime := W1202_USedTime + Cycle_Time; END_IF
IF fbW1210.OUT_TWC <> 0 THEN W1202_USedTime := W1202_USedTime + Cycle_Time; END_IF
IF fbW1212.OUT_TWC <> 0 THEN W1202_USedTime := W1202_USedTime + Cycle_Time; END_IF
IF fbW1214.OUT_TWC <> 0 THEN W1202_USedTime := W1202_USedTime + Cycle_Time; END_IF
IF fbW1602.OUT_TWC <> 0 THEN W1202_USedTime := W1202_USedTime + Cycle_Time; END_IF
IF fbW1604.OUT_TWC <> 0 THEN W1202_USedTime := W1202_USedTime + Cycle_Time; END_IF


(*Save Persistent Vars when power down*)
(*fbUPS();*)
END_PROGRAM

(* POU FB/FB_SE_CYLINDER_POS, ST *)
FUNCTION_BLOCK FB_SE_CYLINDER_POS
VAR_INPUT
	Enable : BOOL;
	Ready  : BOOL;

	IN_CylIn  : ARRAY[1..2] OF BOOL;
	IN_CylOut : ARRAY[1..2] OF BOOL;

	IN_RemIn  : BOOL;
	IN_RemOut : BOOL;
END_VAR
VAR_IN_OUT
	P   : ST_SENSOR_BAR;
	LS  : ST_SENSOR_POS;
	CFG : ST_SE_CYLINDER_POS_CFG;
END_VAR
VAR_OUTPUT
	OUT_CylIn  : BOOL;
	OUT_CylOut : BOOL;

	OUT_Ease   : REAL;

	OUT_HP     : BYTE;
END_VAR
VAR
	State   : WORD;

	IN_Hmi_CylIn  : BOOL;
	IN_Hmi_CylOut : BOOL;

	SIIn  : ARRAY[1..4] OF FB_SMART_INPUT;
	SIOut : ARRAY[1..4] OF FB_SMART_INPUT;

	EventIn  : EN_SMART_INPUT_STATE;
	EventOut : EN_SMART_INPUT_STATE;

	TimeCnt : REAL;
	TimeOut : BOOL;

	LS_In   : BOOL;
	LS_Out  : BOOL;

	ToFaroValue : REAL;
END_VAR
LS_Out := LS.Pos > CFG.TgtLS_Out;
LS_In  := LS.Pos < CFG.TgtLS_In;

(*Check Inputs*)
SIIn[1](In:= IN_CylIn[1],  T_Cont:= T#0ms, T_DClk:= T#0ms);
SIIn[2](In:= IN_CylIn[2],  T_Cont:= T#0ms, T_DClk:= T#0ms);
SIIn[3](In:= IN_Hmi_CylIn, T_Cont:= T#0ms, T_DClk:= T#0ms);
SIIn[4](In:= IN_RemIn,     T_Cont:= T#0ms, T_DClk:= T#0ms);

SIOut[1](In:= IN_CylOut[1],  T_Cont:= T#0ms, T_DClk:= T#0ms);
SIOut[2](In:= IN_CylOut[2],  T_Cont:= T#0ms, T_DClk:= T#0ms);
SIOut[3](In:= IN_Hmi_CylOut, T_Cont:= T#0ms, T_DClk:= T#0ms);
SIOut[4](In:= IN_RemOut,     T_Cont:= T#0ms, T_DClk:= T#0ms);

IF NOT Enable THEN
	OUT_CylIn  := FALSE;
	OUT_CylOut := FALSE;
	OUT_Ease   := 0.0;
	OUT_HP     := 0;

	ToFaroValue := 0.0;

	TimeCnt := 0.0;
	State   := 0;
	RETURN;
END_IF

(*Check Time*)
TimeOut := TimeOut OR ( CFG.TimeMax > 0  AND TimeCnt > CFG.TimeMax );
TimeCnt := TimeCnt + CFG.Cycle;

IF    SIIn[1].Event <> NONE THEN EventIn := SIIn[1].Event;
ELSIF SIIn[2].Event <> NONE THEN EventIn := SIIn[2].Event;
ELSIF SIIn[3].Event <> NONE THEN EventIn := SIIn[3].Event;
ELSIF SIIn[4].Event <> NONE THEN EventIn := SIIn[4].Event;
ELSE
	EventIn := NONE;
END_IF

IF    SIOut[1].Event <> NONE THEN EventOut := SIOut[1].Event;
ELSIF SIOut[2].Event <> NONE THEN EventOut := SIOut[2].Event;
ELSIF SIOut[3].Event <> NONE THEN EventOut := SIOut[3].Event;
ELSIF SIOut[4].Event <> NONE THEN EventOut := SIOut[4].Event;
ELSE
	EventOut := NONE;
END_IF

(*Working States*)
CASE State OF

(*Init State*)
0:
	ToFaroValue := 0.0;

	(*Start Manual IN*)
	IF EventIn = INIT_CONTINUOUS AND Ready AND NOT P.AlMax AND NOT (CFG.LS_Limit_In AND (LS_In OR LS.Err)) THEN
		OUT_CylIn  := TRUE;
		OUT_CylOut := FALSE;
		OUT_Ease   := 0.0;

	    IF LS.Pos < CFG.TgtLS_Slow
		THEN OUT_HP := 1;
		ELSE OUT_HP := CFG.HP;
		END_IF

		TimeOut := FALSE; (*Reset TimeOut Error*)
		State   := 1100;  (*Next State*)

		ToFaroValue := 1.0;

	(*Start Manual OUT*)
	ELSIF EventOut = INIT_CONTINUOUS AND NOT (CFG.LS_Limit_Out AND (LS_Out OR LS.Err)) THEN
		OUT_CylIn  := FALSE;
		OUT_CylOut := TRUE;
		OUT_Ease   := CFG.Ease;
		OUT_HP     := 0;

		TimeOut := FALSE; (*Reset TimeOut Error*)
		State   := 2100;  (*Next State*)

		ToFaroValue := -1.0;

	(*Nothing*)
	ELSE
		OUT_CylIn  := FALSE;
		OUT_CylOut := FALSE;
		OUT_Ease   := 0.0;
		OUT_HP     := 0;

	END_IF

    TimeCnt := 0.0; (*Time Count*)

(*Manual IN*)
1100:
	(*End IN*)
	IF EventIn <> NONE OR EventOut <> NONE OR TimeOut OR P.AlMax OR CFG.LS_Limit_In AND (LS_In OR LS.Err) THEN
		OUT_CylIn  := FALSE;
		OUT_CylOut := FALSE;
		OUT_Ease   := 0.0;
		OUT_HP     := 0;

		State := 0; (*Next State*)

	ELSIF LS.Pos < CFG.TgtLS_Slow THEN
		OUT_HP     := 1;

	END_IF

(*Manual OUT*)
2100:
	(*End OUT*)
	IF EventOut <> NONE OR EventIn <> NONE OR TimeOut OR CFG.LS_Limit_Out AND (LS_Out OR LS.Err)THEN
		OUT_CylIn  := FALSE;
		OUT_CylOut := FALSE;
		OUT_Ease   := 0.0;
		OUT_HP     := 0;

		State := 0; (*Next State*)

	ELSIF TimeCnt > CFG.TimeEase THEN
		OUT_Ease   := 0.0;

	END_IF

END_CASE
END_FUNCTION_BLOCK

(* POU FB/FB_DE_CYLINDER, ST *)
FUNCTION_BLOCK FB_DE_CYLINDER
VAR_INPUT
	Enable : BOOL;
	Ready  : BOOL;

	IN_CylIn  : ARRAY[1..2] OF BOOL;
	IN_CylOut : ARRAY[1..2] OF BOOL;
END_VAR
VAR_IN_OUT
	P_In  : ST_SENSOR_BAR;
	P_Out : ST_SENSOR_BAR;
	CFG   : ST_SE_CYLINDER_CFG;
END_VAR
VAR_OUTPUT
	OUT_CylIn  : BOOL;
	OUT_CylOut : BOOL;
	OUT_Ease   : REAL;
	OUT_HP     : BYTE;
END_VAR
VAR
	State   : WORD;

	IN_Hmi_CylIn  : BOOL;
	IN_Hmi_CylOut : BOOL;

	SIIn  : ARRAY[1..3] OF FB_SMART_INPUT;
	SIOut : ARRAY[1..3] OF FB_SMART_INPUT;

	EventIn  : EN_SMART_INPUT_STATE;
	EventOut : EN_SMART_INPUT_STATE;

	TimeCnt : REAL;
	TimeOut : BOOL;

	ToFaroValue : REAL;

END_VAR
(*Check Inputs*)
SIIn[1](In:= IN_CylIn[1],  T_Cont:= T#0ms, T_DClk:= T#0ms);
SIIn[2](In:= IN_CylIn[2],  T_Cont:= T#0ms, T_DClk:= T#0ms);
SIIn[3](In:= IN_Hmi_CylIn, T_Cont:= T#0ms, T_DClk:= T#0ms);

SIOut[1](In:= IN_CylOut[1],  T_Cont:= T#0ms, T_DClk:= T#0ms);
SIOut[2](In:= IN_CylOut[2],  T_Cont:= T#0ms, T_DClk:= T#0ms);
SIOut[3](In:= IN_Hmi_CylOut, T_Cont:= T#0ms, T_DClk:= T#0ms);

IF NOT Enable THEN
	OUT_CylIn  := FALSE;
	OUT_CylOut := FALSE;
	OUT_Ease   := 0.0;
	OUT_HP     := 0;

	ToFaroValue := 0.0;

	TimeCnt := 0.0;
	State   := 0;
	RETURN;
END_IF

(*Check Time*)
TimeOut := TimeOut OR ( CFG.TimeMax > 0  AND TimeCnt > CFG.TimeMax );
TimeCnt := TimeCnt + CFG.Cycle;

IF    SIIn[1].Event <> NONE THEN EventIn := SIIn[1].Event;
ELSIF SIIn[2].Event <> NONE THEN EventIn := SIIn[2].Event;
ELSIF SIIn[3].Event <> NONE THEN EventIn := SIIn[3].Event;
ELSE
	EventIn := NONE;
END_IF

IF    SIOut[1].Event <> NONE THEN EventOut := SIOut[1].Event;
ELSIF SIOut[2].Event <> NONE THEN EventOut := SIOut[2].Event;
ELSIF SIOut[3].Event <> NONE THEN EventOut := SIOut[3].Event;
ELSE
	EventOut := NONE;
END_IF

(*Working States*)
CASE State OF

(*Init State*)
0:
	ToFaroValue := 0.0;

	(*Start Manual IN*)
	IF EventIn = INIT_CONTINUOUS AND Ready AND NOT P_In.AlMax THEN
		OUT_CylIn  := TRUE;
		OUT_CylOut := FALSE;
		OUT_Ease   := CFG.Ease;
		OUT_HP     := CFG.HP;

		TimeOut := FALSE; (*Reset TimeOut Error*)
		State   := 1100;  (*Next State*)

		ToFaroValue := 1.0;

	(*Start Manual OUT*)
	ELSIF EventOut = INIT_CONTINUOUS AND Ready AND NOT P_Out.AlMax THEN
		OUT_CylIn  := FALSE;
		OUT_CylOut := TRUE;
		OUT_Ease   := CFG.Ease;
		OUT_HP     := CFG.HP;

		TimeOut := FALSE; (*Reset TimeOut Error*)
		State   := 2100;  (*Next State*)

		ToFaroValue := -1.0;

	(*Nothing*)
	ELSE
		OUT_CylIn  := FALSE;
		OUT_CylOut := FALSE;
		OUT_Ease   := 0.0;
		OUT_HP     := 0;

	END_IF

    TimeCnt := 0.0; (*Time Count*)

(*Manual IN*)
1100:
	(*End IN*)
	IF EventIn <> NONE OR EventOut <> NONE OR TimeOut OR P_In.AlMax THEN
		OUT_CylIn  := FALSE;
		OUT_CylOut := FALSE;
		OUT_Ease   := 0.0;
		OUT_HP     := 0;

		State := 0; (*Next State*)

	ELSIF TimeCnt > CFG.TimeEase THEN
		OUT_Ease   := 0.0;

	END_IF

(*Manual OUT*)
2100:
	(*End OUT*)
	IF EventOut <> NONE OR EventIn <> NONE OR TimeOut OR P_Out.AlMax THEN
		OUT_CylIn  := FALSE;
		OUT_CylOut := FALSE;
		OUT_Ease   := 0.0;
		OUT_HP     := 0;

		State := 0; (*Next State*)

	ELSIF TimeCnt > CFG.TimeEase THEN
		OUT_Ease   := 0.0;

	END_IF

END_CASE
END_FUNCTION_BLOCK

(* POU FB/FB_SE_CYLINDER, ST *)
FUNCTION_BLOCK FB_SE_CYLINDER
VAR_INPUT
	Enable : BOOL;
	Ready  : BOOL;

	IN_CylIn  : ARRAY[1..2] OF BOOL;
	IN_CylOut : ARRAY[1..2] OF BOOL;
END_VAR
VAR_IN_OUT
	P   : ST_SENSOR_BAR;
	CFG : ST_SE_CYLINDER_CFG;
END_VAR
VAR_OUTPUT
	OUT_CylIn  : BOOL;
	OUT_CylOut : BOOL;
	OUT_Ease   : REAL;
	OUT_HP     : BYTE;
END_VAR
VAR
	State   : WORD;

	IN_Hmi_CylIn  : BOOL;
	IN_Hmi_CylOut : BOOL;

	SIIn  : ARRAY[1..3] OF FB_SMART_INPUT;
	SIOut : ARRAY[1..3] OF FB_SMART_INPUT;

	EventIn  : EN_SMART_INPUT_STATE;
	EventOut : EN_SMART_INPUT_STATE;

	TimeCnt : REAL;
	TimeOut : BOOL;

	ToFaroValue: REAL;
END_VAR
(*Check Inputs*)
SIIn[1](In:= IN_CylIn[1],  T_Cont:= T#0ms, T_DClk:= T#0ms);
SIIn[2](In:= IN_CylIn[2],  T_Cont:= T#0ms, T_DClk:= T#0ms);
SIIn[3](In:= IN_Hmi_CylIn, T_Cont:= T#0ms, T_DClk:= T#0ms);

SIOut[1](In:= IN_CylOut[1],  T_Cont:= T#0ms, T_DClk:= T#0ms);
SIOut[2](In:= IN_CylOut[2],  T_Cont:= T#0ms, T_DClk:= T#0ms);
SIOut[3](In:= IN_Hmi_CylOut, T_Cont:= T#0ms, T_DClk:= T#0ms);

IF NOT Enable THEN
	OUT_CylIn  := FALSE;
	OUT_CylOut := FALSE;
	OUT_Ease   := 0.0;
	OUT_HP     := 0;

	ToFaroValue := 0.0;

	TimeCnt := 0.0;
	State   := 0;
	RETURN;
END_IF

(*Check Time*)
TimeOut := TimeOut OR ( CFG.TimeMax > 0  AND TimeCnt > CFG.TimeMax );
TimeCnt := TimeCnt + CFG.Cycle;

IF    SIIn[1].Event <> NONE THEN EventIn := SIIn[1].Event;
ELSIF SIIn[2].Event <> NONE THEN EventIn := SIIn[2].Event;
ELSIF SIIn[3].Event <> NONE THEN EventIn := SIIn[3].Event;
ELSE
	EventIn := NONE;
END_IF

IF    SIOut[1].Event <> NONE THEN EventOut := SIOut[1].Event;
ELSIF SIOut[2].Event <> NONE THEN EventOut := SIOut[2].Event;
ELSIF SIOut[3].Event <> NONE THEN EventOut := SIOut[3].Event;
ELSE
	EventOut := NONE;
END_IF

(*Working States*)
CASE State OF

(*Init State*)
0:
	ToFaroValue := 0.0;

	(*Start Manual IN*)
	IF EventIn = INIT_CONTINUOUS AND Ready AND NOT P.AlMax THEN
		OUT_CylIn  := TRUE;
		OUT_CylOut := FALSE;
		OUT_Ease   := 0.0;
		OUT_HP     := CFG.HP;

		TimeOut := FALSE; (*Reset TimeOut Error*)
		State   := 1100;  (*Next State*)

		ToFaroValue := 1.0;

	(*Start Manual OUT*)
	ELSIF EventOut = INIT_CONTINUOUS THEN
		OUT_CylIn  := FALSE;
		OUT_CylOut := TRUE;
		OUT_Ease   := CFG.Ease;
		OUT_HP     := 0;

		TimeOut := FALSE; (*Reset TimeOut Error*)
		State   := 2100;  (*Next State*)

		ToFaroValue := -1.0;

	(*Nothing*)
	ELSE
		OUT_CylIn  := FALSE;
		OUT_CylOut := FALSE;
		OUT_Ease   := 0.0;
		OUT_HP     := 0;

	END_IF

    TimeCnt := 0.0; (*Time Count*)

(*Manual IN*)
1100:
	(*End IN*)
	IF EventIn <> NONE OR EventOut <> NONE OR TimeOut OR P.AlMax THEN
		OUT_CylIn  := FALSE;
		OUT_CylOut := FALSE;
		OUT_Ease   := 0.0;
		OUT_HP     := 0;

		State := 0; (*Next State*)

	END_IF

(*Manual OUT*)
2100:
	(*End OUT*)
	IF EventOut <> NONE OR EventIn <> NONE OR TimeOut THEN
		OUT_CylIn  := FALSE;
		OUT_CylOut := FALSE;
		OUT_Ease   := 0.0;
		OUT_HP     := 0;

		State := 0; (*Next State*)

	ELSIF TimeCnt > CFG.TimeEase THEN
		OUT_Ease   := 0.0;

	END_IF

END_CASE
END_FUNCTION_BLOCK

(* POU FB/FB_SE_CYLINDER_QR, ST *)
FUNCTION_BLOCK FB_SE_CYLINDER_QR
VAR_INPUT
	Enable : BOOL;
	Ready  : BOOL;

	IN_CylIn  : ARRAY[1..2] OF BOOL;
	IN_CylOut : ARRAY[1..2] OF BOOL;
	IN_CylQR  : ARRAY[1..2] OF BOOL;
END_VAR
VAR_IN_OUT
	P   : ST_SENSOR_BAR;
	CFG : ST_SE_CYLINDER_CFG;
END_VAR
VAR_OUTPUT
	OUT_CylIn  : BOOL;
	OUT_CylOut : BOOL;
	OUT_Ease   : REAL;
	OUT_HP     : BYTE;
END_VAR
VAR
	State   : WORD;

	IN_Hmi_CylIn  : BOOL;
	IN_Hmi_CylOut : BOOL;
	IN_Hmi_CylQR  : BOOL;

	SIIn  : ARRAY[1..3] OF FB_SMART_INPUT;
	SIOut : ARRAY[1..3] OF FB_SMART_INPUT;
	SIQR  : ARRAY[1..3] OF FB_SMART_INPUT;

	EventIn  : EN_SMART_INPUT_STATE;
	EventOut : EN_SMART_INPUT_STATE;
	EventQR  : EN_SMART_INPUT_STATE;

	TimeCnt : REAL;
	TimeOut : BOOL;

	ToFaroValue : REAL;
END_VAR
(*Check Inputs*)
SIIn[1](In:= IN_CylIn[1],  T_Cont:= T#0ms, T_DClk:= T#0ms);
SIIn[2](In:= IN_CylIn[2],  T_Cont:= T#0ms, T_DClk:= T#0ms);
SIIn[3](In:= IN_Hmi_CylIn, T_Cont:= T#0ms, T_DClk:= T#0ms);

SIOut[1](In:= IN_CylOut[1],  T_Cont:= T#0ms, T_DClk:= T#0ms);
SIOut[2](In:= IN_CylOut[2],  T_Cont:= T#0ms, T_DClk:= T#0ms);
SIOut[3](In:= IN_Hmi_CylOut, T_Cont:= T#0ms, T_DClk:= T#0ms);

SIQR[1](In:= IN_CylQR[1],  T_Cont:= T#0ms, T_DClk:= T#0ms);
SIQR[2](In:= IN_CylQR[2],  T_Cont:= T#0ms, T_DClk:= T#0ms);
SIQR[3](In:= IN_Hmi_CylQR, T_Cont:= T#0ms, T_DClk:= T#0ms);

IF NOT Enable THEN
	OUT_CylIn  := FALSE;
	OUT_CylOut := FALSE;
	OUT_Ease   := 0.0;
	OUT_HP     := 0;

	ToFaroValue := 0.0;

	TimeCnt := 0.0;
	State   := 0;
	RETURN;
END_IF

(*Check Time*)
TimeOut := TimeOut OR ( CFG.TimeMax > 0  AND TimeCnt > CFG.TimeMax);
TimeCnt := TimeCnt + 1;

IF    SIIn[1].Event <> NONE THEN EventIn := SIIn[1].Event;
ELSIF SIIn[2].Event <> NONE THEN EventIn := SIIn[2].Event;
ELSIF SIIn[3].Event <> NONE THEN EventIn := SIIn[3].Event;
ELSE
	EventIn := NONE;
END_IF

IF    SIOut[1].Event <> NONE THEN EventOut := SIOut[1].Event;
ELSIF SIOut[2].Event <> NONE THEN EventOut := SIOut[2].Event;
ELSIF SIOut[3].Event <> NONE THEN EventOut := SIOut[3].Event;
ELSE
	EventOut := NONE;
END_IF

IF    SIQR[1].Event <> NONE THEN EventQR := SIQR[1].Event;
ELSIF SIQR[2].Event <> NONE THEN EventQR := SIQR[2].Event;
ELSIF SIQR[3].Event <> NONE THEN EventQR := SIQR[3].Event;
ELSE
	EventQR := NONE;
END_IF

(*Working States*)
CASE State OF

(*Init State*)
0:
	ToFaroValue := 0.0;

	(*Start Manual IN*)
	IF EventIn = INIT_CONTINUOUS AND Ready AND NOT P.AlMax THEN
		OUT_CylIn  := TRUE;
		OUT_CylOut := FALSE;
		OUT_Ease   := 0.0;
		OUT_HP     := Cfg.HP;

		TimeOut := FALSE; (*Reset TimeOut Error*)
		State   := 1100;  (*Next State*)

		ToFaroValue := 1.0;

	(*Start Manual OUT*)
	ELSIF EventOut = INIT_CONTINUOUS THEN
		OUT_CylIn  := FALSE;
		OUT_CylOut := TRUE;
		OUT_Ease   := Cfg.Ease;
		OUT_HP     := 0;

		TimeOut := FALSE; (*Reset TimeOut Error*)
		State   := 2100;  (*Next State*)

		ToFaroValue := -1.0;

	(*Start QR OUT*)
	ELSIF EventQR = INIT_CONTINUOUS THEN
		OUT_CylIn  := FALSE;
		OUT_CylOut := TRUE;
		OUT_Ease   := 0.0;
		OUT_HP     := 0;

		TimeOut := FALSE; (*Reset TimeOut Error*)
		State   := 2200;  (*Next State*)

		ToFaroValue := -2.0;

	(*Nothing*)
	ELSE
		OUT_CylIn  := FALSE;
		OUT_CylOut := FALSE;
		OUT_Ease   := 0.0;
		OUT_HP     := 0;

	END_IF

    TimeCnt := 0; (*Time Count*)

(*Manual IN*)
1100:
	(*End IN*)
	IF EventIn <> NONE OR EventOut <> NONE OR TimeOut OR P.AlMax THEN
		OUT_CylIn  := FALSE;
		OUT_CylOut := FALSE;
		OUT_Ease   := 0.0;
		OUT_HP     := 0;

		State := 0; (*Next State*)

	(*Start QR OUT*)
	ELSIF EventQR = INIT_CONTINUOUS THEN
		OUT_CylIn  := FALSE;
		OUT_CylOut := TRUE;
		OUT_Ease   := 0.0;
		OUT_HP     := 0;

		TimeCnt := 0;    (*Time Count*)
		State   := 2200; (*Next State*)

		ToFaroValue := -2.0;

	END_IF

(*Manual OUT*)
2100:
	(*End OUT*)
	IF EventOut <> NONE OR EventIn <> NONE OR TimeOut THEN
		OUT_CylIn  := FALSE;
		OUT_CylOut := FALSE;
		OUT_Ease   := 0.0;
		OUT_HP     := 0;

		State := 0; (*Next State*)

	(*Start QR OUT*)
	ELSIF EventQR = INIT_CONTINUOUS THEN
		OUT_CylIn  := FALSE;
		OUT_CylOut := TRUE;
		OUT_Ease   := 0.0;
		OUT_HP     := 0;

		TimeCnt := 0;    (*Time Count*)
		State   := 2200; (*Next State*)

		ToFaroValue := -2.0;

	ELSIF TimeCnt > CFG.TimeEase THEN
		OUT_Ease   := 0.0;

	END_IF

(*QR OUT*)
2200:
	(*End QR OUT*)
	IF EventQR <> NONE OR TimeOut THEN
		OUT_CylIn  := FALSE;
		OUT_CylOut := FALSE;
		OUT_Ease   := 0.0;
		OUT_HP     := 0;

		State := 0; (*Next State*)
	END_IF

END_CASE
END_FUNCTION_BLOCK

(* POU FB/FB_LIFTING_PROPELLER, ST *)
FUNCTION_BLOCK FB_LIFTING_PROPELLER
VAR_INPUT
	Enable  : BOOL;
	ReadyUp : BOOL;
	Clear   : BOOL;

	IN_CylIn  : ARRAY[1..2] OF BOOL; (*Up*)
	IN_CylOut : ARRAY[1..2] OF BOOL; (*Dw*)
END_VAR
VAR_IN_OUT
	P_In  : ST_SENSOR_BAR;
	P_Out : ST_SENSOR_BAR;
	LS    : ST_SENSOR_POS;
	CFG   : ST_LIFT_PROP_CFG;
END_VAR
VAR_OUTPUT
	OUT_EV1 : BOOL; (*Pump OUT*)
	OUT_EV2 : BOOL; (*Ease OUT*)
	OUT_EV3 : BOOL; (*Pump IN*)
	OUT_EV4 : BOOL; (*Ease IN*)

	OUT_HP  : BYTE;

	PROP_UP : BOOL;
	PROP_DW : BOOL;
END_VAR
VAR
	State   : WORD;

	IN_Hmi_CylIn  : BOOL;
	IN_Hmi_CylOut : BOOL;

	SIIn  : ARRAY[1..3] OF FB_SMART_INPUT;
	SIOut : ARRAY[1..3] OF FB_SMART_INPUT;

	EventIn  : EN_SMART_INPUT_STATE;
	EventOut : EN_SMART_INPUT_STATE;

	TimeCnt : REAL;
	TimeOut : BOOL;

	P_Bypass  : BOOL;

	Slow : BOOL;
	LS_Dif : REAL;

	LS_Up : BOOL;
	LS_Dw : BOOL;
	P_Up : BOOL;
	P_Dw : BOOL;

	Alarm : ST_Alarm;

	ToFaroValue : REAL;

END_VAR
VAR PERSISTENT
	Man_Up AT %Q*: BOOL;
	Man_Dw AT %Q*: BOOL;
END_VAR
IF Clear THEN
	Alarm.Alarm := FALSE;
	Alarm.Adver := FALSE;
	Alarm.AlCnt := 0;
	Alarm.AlLen := 0.0;
END_IF

LS_Dw := NOT LS.Err AND LS.Pos > CFG.TgtLS_Dw - CFG.LS_DB;
LS_Up := NOT LS.Err AND LS.Pos < CFG.TgtLS_Up + CFG.LS_DB;
P_Dw  := NOT P_Out.Err AND P_Out.Bar > CFG.TgtP_Dw - CFG.P_DB;
P_Up  := NOT P_In.Err  AND P_In.Bar  > CFG.TgtP_Up - CFG.P_DB;

(*Check Inputs*)
SIIn[1](In:= IN_CylIn[1],  T_Cont:= T#500ms, T_DClk:= T#0ms);
SIIn[2](In:= IN_CylIn[2],  T_Cont:= T#500ms, T_DClk:= T#0ms);
SIIn[3](In:= IN_Hmi_CylIn, T_Cont:= T#500ms, T_DClk:= T#0ms);

SIOut[1](In:= IN_CylOut[1],  T_Cont:= T#500ms, T_DClk:= T#0ms);
SIOut[2](In:= IN_CylOut[2],  T_Cont:= T#500ms, T_DClk:= T#0ms);
SIOut[3](In:= IN_Hmi_CylOut, T_Cont:= T#500ms, T_DClk:= T#0ms);

IF NOT Enable THEN
	OUT_EV1 := FALSE;
	OUT_EV2 := FALSE;
	OUT_EV3 := FALSE;
	OUT_EV4 := FALSE;

	OUT_HP   := 0;

	PROP_UP := FALSE;
	PROP_DW := FALSE;

	ToFaroValue := 0.0;

	Alarm.Alarm := FALSE;
	Alarm.Adver := FALSE;
	Alarm.AlCnt := 0;
	Alarm.AlLen := 0.0;

	TimeCnt := 0.0;
	State   := 0;
	RETURN;
END_IF

(*Check Time*)
TimeOut := TimeOut OR ( CFG.TimeMax > 0  AND TimeCnt > CFG.TimeMax );
TimeCnt := TimeCnt + CFG.Cycle;

IF    SIIn[1].Event <> NONE THEN EventIn := SIIn[1].Event;
ELSIF SIIn[2].Event <> NONE THEN EventIn := SIIn[2].Event;
ELSIF SIIn[3].Event <> NONE THEN EventIn := SIIn[3].Event;
ELSE							 EventIn := NONE;
END_IF

IF    SIOut[1].Event <> NONE THEN EventOut := SIOut[1].Event;
ELSIF SIOut[2].Event <> NONE THEN EventOut := SIOut[2].Event;
ELSIF SIOut[3].Event <> NONE THEN EventOut := SIOut[3].Event;
ELSE							  EventOut := NONE;
END_IF

(*Working States*)
CASE State OF

(*Init State*)
0:
	OUT_EV1 := FALSE;
	OUT_EV2 := FALSE;
	OUT_EV3 := FALSE;
	OUT_EV4 := FALSE;
	OUT_HP  := 0;

    TimeCnt  := 0.0; (*Time Count*)

	ToFaroValue := 0.0;

	(*Start Manual IN/UP*)
	IF EventIn = INIT_CONTINUOUS AND ReadyUp THEN
		(*PROP_UP := FALSE;*)
		PROP_DW := FALSE;
		TimeOut := FALSE;

		(*Next State*)
		IF LS.Err OR Man_Up OR Man_Dw
		THEN State := 100;
		ELSE State := 110;
		END_IF

		ToFaroValue := 1.0;

	(*Start Manual OUT/DW*)
	ELSIF EventOut = INIT_CONTINUOUS THEN
		PROP_UP := FALSE;
		(*PROP_DW := FALSE;*)
		TimeOut := FALSE;

		(*Next State*)
		IF LS.Err OR Man_Up OR Man_Dw
		THEN State := 200;
		ELSE State := 210;
		END_IF

		ToFaroValue := -1.0;

	ELSE
		(*Override mode*)
		IF Man_Up OR Man_Dw THEN
			Man_Dw := Man_Dw AND NOT Man_Up;

			PROP_UP := Man_Up;
			PROP_DW := Man_Dw;

			IF Man_Up THEN Alarm.Adver := TRUE; Alarm.Text := 'Propulsion Up/Dw. Manual Override UP Position.'; END_IF
			IF Man_Dw THEN Alarm.Adver := TRUE; Alarm.Text := 'Propulsion Up/Dw. Manual Override DW Position.'; END_IF

		(*Init state *)
		ELSIF NOT PROP_UP AND NOT PROP_DW THEN
			PROP_UP := LS_Up AND P_Up;
			PROP_DW := LS_Dw AND P_Dw;

			(*Alarm := LS.Err;*)

		ELSE
			(*Prevent propulsion OFF in case of sensors problem*)
			IF PROP_DW THEN

				IF NOT P_Dw  THEN Alarm.Adver := TRUE; Alarm.Text :=  '(P601) Propulsion Up/Dw. Missing DW Press. Target.';   END_IF

				IF NOT LS_Dw THEN
					IF NOT Alarm.Alarm THEN
						Alarm.AlCnt  := Alarm.AlCnt + 1;
						Alarm.AlLen  := 0.0;
						Alarm.TimeInit := INPUTS.sLocal;
						Alarm.AlInit   := TRUE;

					ELSE
						Alarm.AlLen  := Alarm.AlLen + MAIN.Cycle_Time;

					END_IF

					Alarm.Adver := TRUE;
					Alarm.Alarm := TRUE;

					Alarm.Text  := '(LS601) Propulsion Up/Dw. Missing DW Position Target.';

				ELSE
					IF Alarm.Alarm THEN
						Alarm.TimeEnd := INPUTS.sLocal;
						Alarm.AlEnd   := TRUE;

					END_IF

					Alarm.Alarm := FALSE;

				END_IF

			END_IF

			IF PROP_UP THEN
				IF NOT P_Up  THEN Alarm.Adver := TRUE; Alarm.Text :=  '(P603) Propulsion Up/Dw. Missing UP Press. Target.';   END_IF
				IF NOT LS_Up THEN Alarm.Adver := TRUE; Alarm.Text := '(LS601) Propulsion Up/Dw. Missing UP Position Target.'; END_IF
			END_IF

		END_IF

	END_IF

	IF NOT PROP_DW THEN
		IF Alarm.Alarm THEN
			Alarm.TimeEnd := INPUTS.sLocal;
			Alarm.AlEnd   := TRUE;

		END_IF

		Alarm.Alarm := FALSE;

	END_IF


(*** MANUAL ***)
(*IN/UP*)
100:
	IF EventIn = END_CONTINUOUS OR EventOut <> NONE OR NOT ReadyUp OR TimeOut OR P_In.AlMax THEN
		Out_HP := 0;
		State  := 0;  (*Next State*)

	ELSE
		OUT_EV1 := FALSE;
		OUT_EV2 := TRUE;
		OUT_EV3 := TRUE;
		OUT_EV4 := FALSE;

		OUT_HP := 1; (*Manual Slow*)
		Slow   := TRUE;

	END_IF

(*** AUTO ***)
(*Pumping IN/UP*)
110:
	IF EventIn = END_CONTINUOUS OR EventOut <> NONE OR NOT ReadyUp OR TimeOut OR LS.Err OR Man_Up OR Man_Dw OR P_In.AlMax THEN
		OUT_HP := 0;
		State  := 0;  (*Next State*)

	ELSIF LS.Pos <= CFG.TgtLS_Up THEN
		OUT_EV1 := FALSE;
		OUT_EV2 := FALSE; (*Close to presurize*)
		OUT_EV3 := TRUE;
		OUT_EV4 := FALSE;

		OUT_HP := 1; (*Slow*)
		Slow   := TRUE;
		State  := 120;

	ELSIF (LS.Pos - CFG.TgtLS_Up) < CFG.LS_DB THEN
		OUT_EV1 := FALSE;
		OUT_EV2 := TRUE;
		OUT_EV3 := TRUE;
		OUT_EV4 := FALSE;

		OUT_HP := 1; (*Slow*)
		Slow   := TRUE;

	ELSE
		OUT_EV1 := FALSE;
		OUT_EV2 := TRUE;
		OUT_EV3 := TRUE;
		OUT_EV4 := FALSE;

		OUT_HP := CFG.HP_Up;
		Slow   := FALSE;

	END_IF

(*Pressurize IN/UP *)
120:
	IF EventIn = END_CONTINUOUS OR EventOut <> NONE OR NOT ReadyUp OR TimeOut OR LS.Err OR Man_Up OR Man_Dw OR P_In.AlMax THEN
		OUT_HP := 0;
		State  := 0;  (*Next State*)

	ELSIF P_In.Bar > CFG.TgtP_Up OR P_In.AlErr THEN
		TimeCnt := 0.0;
		State   := 130;

	END_IF

(*Delay IN/UP *)
130:
	IF EventIn = END_CONTINUOUS OR EventOut <> NONE OR NOT ReadyUp OR TimeOut OR LS.Err OR Man_Up OR Man_Dw OR P_In.AlMax THEN
		OUT_HP := 0;
		State  := 0;  (*Next State*)

	ELSIF TimeCnt > CFG.Delay_Up THEN
		PROP_UP := TRUE;
		OUT_EV3 := FALSE;
		OUT_HP  := 0;
		State   := 0;

	END_IF

(*** MANUAL ***)
(*OUT/DW*)
200:
	IF EventOut = END_CONTINUOUS OR EventIn <> NONE OR TimeOut OR P_Out.AlMax THEN (*OR NOT Ready*)
		OUT_HP := 0;
		State  := 0;  (*Next State*)

	ELSE
		OUT_EV1 := TRUE;
		OUT_EV2 := FALSE;
		OUT_EV3 := FALSE;
		OUT_EV4 := TRUE;

		OUT_HP := 1;
		Slow   := TRUE;
	END_IF

(*** AUTO ***)
(*Pumping OUT/DW*)
210:
	IF EventOut = END_CONTINUOUS OR EventIn <> NONE OR TimeOut OR LS.Err OR Man_Up OR Man_Dw OR P_Out.AlMax THEN (*OR NOT Ready*)
		OUT_HP := 0;
		State  := 0;  (*Next State*)

	ELSIF LS.Pos >= CFG.TgtLS_Dw THEN
		PROP_DW := TRUE; (*Better activate here*)

		OUT_EV1 := TRUE;
		OUT_EV2 := FALSE;
		OUT_EV3 := FALSE;
		OUT_EV4 := FALSE; (*Close to presurize*)

		OUT_HP := 1; (*Slow*)
		Slow   := TRUE;
		State  := 220;

	ELSIF (CFG.TgtLS_Dw - LS.Pos) < CFG.LS_DB THEN
		OUT_EV1 := TRUE;
		OUT_EV2 := FALSE;
		OUT_EV3 := FALSE;
		OUT_EV4 := TRUE;

		OUT_HP := 1; (*Slow*)
		Slow   := TRUE;

	ELSE
		OUT_EV1 := TRUE;
		OUT_EV2 := FALSE;
		OUT_EV3 := FALSE;
		OUT_EV4 := TRUE;

		OUT_HP := CFG.HP_Dw;
		Slow   := FALSE;

	END_IF

(*Pressurize OUT/DW *)
220:
	IF EventOut = END_CONTINUOUS OR EventIn <> NONE OR TimeOut OR LS.Err OR Man_Up OR Man_Dw OR P_Out.AlMax THEN (*OR NOT Ready*)
		OUT_HP := 0;
		State  := 0;  (*Next State*)

	ELSIF P_Out.Bar > CFG.TgtP_Dw OR P_Out.Err THEN
		PROP_DW := TRUE;
		TimeCnt := 0.0;
		State   := 230;

	END_IF

(*Delay OUT/DW *)
230:
	IF EventOut = END_CONTINUOUS OR EventIn <> NONE OR TimeOut OR LS.Err OR Man_Up OR Man_Dw OR P_Out.AlMax THEN (*OR NOT Ready*)
		OUT_HP := 0;
		State  := 0;  (*Next State*)

	ELSIF TimeCnt > CFG.Delay_Dw THEN
		PROP_DW := TRUE;
		OUT_EV1 := FALSE;
		OUT_HP  := 0;
		State   := 0;

	END_IF

END_CASE
END_FUNCTION_BLOCK

(* POU INPUTS, ST *)
PROGRAM INPUTS
VAR
(*Analog Inputs*)
	(*Node00*)
	Prop_DynRPM : FB_DYN_RPM;

	THR1_Prop_V : FB_AVG5;
	THR2_Prop_V : FB_AVG5;
	THR_Prop_Chk : REAL;

	THR_Alarm : ST_ALARM;

(*Cylinders Buttons*)
	B301 : ARRAY[1..2] OF BOOL;
	B302 : ARRAY[1..2] OF BOOL;
	B303 : ARRAY[1..2] OF BOOL;
	B304 : ARRAY[1..2] OF BOOL;
	B305 : ARRAY[1..2] OF BOOL;
	B306 : ARRAY[1..2] OF BOOL;
	B307 : ARRAY[1..2] OF BOOL;
	B308 : ARRAY[1..2] OF BOOL;
	B309 : ARRAY[1..2] OF BOOL;
	B310 : ARRAY[1..2] OF BOOL;
	B311 : ARRAY[1..2] OF BOOL;
	B312 : ARRAY[1..2] OF BOOL;

	B501 : ARRAY[1..2] OF BOOL;
	B502 : ARRAY[1..2] OF BOOL;
	B503 : ARRAY[1..2] OF BOOL;
	B504 : ARRAY[1..2] OF BOOL;
	B505 : ARRAY[1..2] OF BOOL;
	B506 : ARRAY[1..2] OF BOOL;
	B506Q: ARRAY[1..2] OF BOOL;

	B601 : ARRAY[1..2] OF BOOL;
	B603 : ARRAY[1..2] OF BOOL;
	B605 : ARRAY[1..2] OF BOOL;
	B607 : ARRAY[1..2] OF BOOL;
	B606 : ARRAY[1..2] OF BOOL;

	B701 : ARRAY[1..2] OF BOOL;
	B702 : ARRAY[1..2] OF BOOL;
	B703 : ARRAY[1..2] OF BOOL;
	B704 : ARRAY[1..2] OF BOOL;
	B705 : ARRAY[1..2] OF BOOL;
	B706 : ARRAY[1..2] OF BOOL;
	B707 : ARRAY[1..2] OF BOOL;
	B708 : ARRAY[1..2] OF BOOL;
	B709 : ARRAY[1..2] OF BOOL;
	B710 : ARRAY[1..2] OF BOOL;

	B901 : ARRAY[1..2] OF BOOL;
	B902 : ARRAY[1..2] OF BOOL;
	B903 : ARRAY[1..2] OF BOOL;
	B904 : ARRAY[1..2] OF BOOL;
	B90T : ARRAY[1..2] OF BOOL;

	BTravA : ARRAY[1..3] OF BOOL;
	BTravB : ARRAY[1..3] OF BOOL;
	BTravT : ARRAY[1..2] OF BOOL;
	BTravD : ARRAY[1..2] OF BOOL;

	BKeelP : ARRAY[1..4] OF BOOL;
	BKeelS : ARRAY[1..4] OF BOOL;
	BKeelC : ARRAY[1..4] OF BOOL;
	BKeelF : ARRAY[1..4] OF BOOL;
	BKeelT : ARRAY[1..2] OF BOOL;

	BBoardP : ARRAY[1..2] OF BOOL;
	BBoardS : ARRAY[1..2] OF BOOL;
	BBoardC : ARRAY[1..2] OF BOOL;

	BBowThrP : BOOL;
	BBowThrS : BOOL;
	BBowThrU : BOOL;
	BBowThrD : BOOL;

	BWB_P_Fwd : ARRAY[1..2] OF BOOL;
	BWB_P_Aft : ARRAY[1..2] OF BOOL;
	BWB_S_Fwd : ARRAY[1..2] OF BOOL;
	BWB_S_Aft : ARRAY[1..2] OF BOOL;
	BWB_Fill  : ARRAY[1..2] OF BOOL;
	BWB_12    : ARRAY[1..2] OF BOOL;
	BWB_Dump  : ARRAY[1..2] OF BOOL;
	BWB_Move  : ARRAY[1..2] OF BOOL;
	BWB_Stop  : ARRAY[1..2] OF BOOL;

	L_Red_Trig    : R_TRIG;
	L_Anchor_Trig : R_TRIG;
	L_Steam_Trig  : R_TRIG;
	L_Deck_Trig   : R_TRIG;
	L_Nav_Trig    : R_TRIG;

	L_HMI_Red_Trig    : R_TRIG;
	L_HMI_Anchor_Trig : R_TRIG;
	L_HMI_Steam_Trig  : R_TRIG;
	L_HMI_Deck_Trig   : R_TRIG;
	L_HMI_Nav_Trig    : R_TRIG;

	Override_Trig : R_TRIG;
	RemPort_Trig  : R_TRIG;
	RemStbd_Trig  : R_TRIG;
	RemOff_Trig   : R_TRIG;

	Override_ON : BOOL;
	RemPort_ON : BOOL;
	RemStbd_ON : BOOL;


(*	N02_IN_BTrig : R_TRIG;
	N03_IN_BTrig : R_TRIG;
	N04_IN_BTrig : R_TRIG;
	N05_IN_BTrig : R_TRIG;
	N06_IN_BTrig : R_TRIG;
	N07_IN_BTrig : R_TRIG;
	N08_IN_BTrig : R_TRIG;
	N09_IN_BTrig : R_TRIG;
	N10_IN_BTrig : R_TRIG;
	N11_IN_BTrig : R_TRIG;
	N12_IN_BTrig : R_TRIG;
	N13_IN_BTrig : R_TRIG;
	N14_IN_BTrig : R_TRIG;
	N15_IN_BTrig : R_TRIG;
	N16_IN_BTrig : R_TRIG;
	N17_IN_BTrig : R_TRIG;
	N18_IN_BTrig : R_TRIG;
	N19_IN_BTrig : R_TRIG;
	N20_IN_BTrig : R_TRIG;
	N21_IN_BTrig : R_TRIG;

	N02_IN_CTrig : R_TRIG;
	N03_IN_CTrig : R_TRIG;
	N04_IN_CTrig : R_TRIG;
	N05_IN_CTrig : R_TRIG;
	N06_IN_Ctrig : R_TRIG;
	N07_IN_Ctrig : R_TRIG;
	N08_IN_CTrig : R_TRIG;
	N09_IN_CTrig : R_TRIG;
	N10_IN_CTrig : R_TRIG;
	N11_IN_CTrig : R_TRIG;
	N12_IN_CTrig : R_TRIG;
	N13_IN_CTrig : R_TRIG;
	N14_IN_CTrig : R_TRIG;
	N15_IN_CTrig : R_TRIG;
	N16_IN_CTrig : R_TRIG;
	N17_IN_CTrig : R_TRIG;
	N18_IN_CTrig : R_TRIG;
	N19_IN_CTrig : R_TRIG;
	N20_IN_CTrig : R_TRIG;
	N21_IN_CTrig : R_TRIG;

	C_PP: BOOL;
	C_PS: BOOL;
	C_SP: BOOL;
	C_SS: BOOL;
	C_MP1: BOOL;
	C_MP2: BOOL;
	C_MS1: BOOL;
	C_MS2: BOOL;*)

	B1202_1 : ARRAY[1..4] OF BOOL;
	B1202_2 : ARRAY[1..4] OF BOOL;
	B1204_1 : ARRAY[1..4] OF BOOL;
	B1204_2 : ARRAY[1..4] OF BOOL;
	B1206_1 : ARRAY[1..4] OF BOOL;
	B1206_2 : ARRAY[1..4] OF BOOL;
	B1208_1 : ARRAY[1..4] OF BOOL;
	B1208_2 : ARRAY[1..4] OF BOOL;
	B1210_1 : ARRAY[1..4] OF BOOL;
	B1210_2 : ARRAY[1..4] OF BOOL;
	B1212_1 : ARRAY[1..4] OF BOOL;
	B1212_2 : ARRAY[1..4] OF BOOL;
	B1214_1 : ARRAY[1..4] OF BOOL;
	B1214_2 : ARRAY[1..4] OF BOOL;

	B1602_1 : ARRAY[1..4] OF BOOL;
	B1602_2 : ARRAY[1..4] OF BOOL;
	B1604_1 : ARRAY[1..4] OF BOOL;
	B1604_2 : ARRAY[1..4] OF BOOL;

	B1202_G : BOOL;
	B1204_G : BOOL;
	B1206_G : BOOL;
	B1208_G : BOOL;
	B1210_G : BOOL;
	B1212_G : BOOL;
	B1214_G : BOOL;

	B1602_G : BOOL;
	B1604_G : BOOL;


(*System Time*)
	fbLocalTime :FB_LocalSystemTime;
	(*tsTime      :TIMESTRUCT;*)
	sLocal      :STRING;
	sVisuTime   :STRING;

END_VAR
(*
Forestay 	= 27500 kg or 525 bar
JibCunn		=  9500 kg or 445 bar
GS			=  4200 kg or 320 bar
Deflector   =  8400 kg or 400 bar
MainCunn	=  2600 kg or 400 bar
Outhaul		=  6500 kg or 450 bar
Vang 		= 19500 kg or 450 bar
JibInOut	=  5500 kg or 470 bar
JibUpDw		=  5000 kg or 440 bar
*)
(*Node00 - PLC*)
Prop_DynRPM( CNT:= N0_CNT1, CycleTime:= 20, MaxWidth:= 500, Accuracy:= 20 );

IF PARAMS.stPropulsionCfg.PropRPM_K > 0
THEN Prop_RPM := Prop_DynRPM.RPM / PARAMS.stPropulsionCfg.PropRPM_K;
ELSE Prop_RPM := Prop_DynRPM.RPM;
END_IF

THR1_Prop_V( IN:= N0_AI1 / 3276.7 );
THR2_Prop_V( IN:= N0_AI2 / 3276.7 );

THR_Prop_Fwd := N0_DI2;
THR_Prop_Rev := N0_DI3;
THR_Prop_Chk := THR1_Prop_V.AVG + THR2_Prop_V.AVG;
THR_Prop_Err := N0_AI1_Err OR THR1_Prop_V.AVG < 0.5 OR THR1_Prop_V.AVG > 4.5
			 OR N0_AI2_Err OR THR2_Prop_V.AVG < 0.5 OR THR2_Prop_V.AVG > 4.5
			 OR THR_Prop_Chk > 5.5 OR THR_Prop_Chk < 4.5;

IF THR_Prop_Fwd THEN
	THR_Prop := THR1_Prop_V.AVG;

ELSIF THR_Prop_Rev THEN
	THR_Prop := -THR1_Prop_V.AVG;

ELSE
	THR_Prop := 0.0;

END_IF

IF ALARMS.Clear THEN
	THR_Alarm.Alarm := FALSE;
	THR_Alarm.Adver := FALSE;
	THR_Alarm.AlCnt := 0;
	THR_Alarm.AlLen := 0.0;

END_IF

IF THR_Prop_Err THEN
	IF NOT THR_Alarm.Alarm THEN
		THR_Alarm.AlCnt  := THR_Alarm.AlCnt + 1;
		THR_Alarm.AlLen  := 0.0;
		THR_Alarm.TimeInit := INPUTS.sLocal;
		THR_Alarm.AlInit   := TRUE;

		THR_Alarm.Text   := 'Propulsion Throttle Error.';

	ELSE
		THR_Alarm.AlLen  := THR_Alarm.AlLen + MAIN.Cycle_Time;

	END_IF

	THR_Alarm.Adver := TRUE;
	THR_Alarm.Alarm := TRUE;

ELSE
	IF THR_Alarm.Alarm THEN
		THR_Alarm.TimeEnd := INPUTS.sLocal;
		THR_Alarm.AlEnd   := TRUE;

	END_IF

	THR_Alarm.Alarm := FALSE;

END_IF

(*SF000 := N0_DI1;*)
F_CALC_SENSOR_NC ( N0_DI1, ALARMS.Clear, MAIN.Cycle_Time, 0.0, SF000 );

(*TANK + GS + MF00 + PP - Node36/37*)
F_CALC_SENSOR_NC ( N37_DI13_CH4_2, ALARMS.Clear, MAIN.Cycle_Time, PARAMS.SF_Delay, SF001 );
F_CALC_SENSOR_NC ( N37_DI9_CH3_2 , ALARMS.Clear, MAIN.Cycle_Time, PARAMS.SF_Delay, SF002 );
F_CALC_SENSOR_NC ( N37_DI5_CH5_2 , ALARMS.Clear, MAIN.Cycle_Time, PARAMS.SF_Delay, SF003 );
F_CALC_SENSOR_NC ( N37_DI1_CH7_2 , ALARMS.Clear, MAIN.Cycle_Time, PARAMS.SF_Delay, SF004 );
F_CALC_SENSOR_NC ( N37_DI3_CH6_2 , ALARMS.Clear, MAIN.Cycle_Time, PARAMS.SF_Delay, SF005 );
F_CALC_SENSOR_NC ( N37_DI7_CH8_2 , ALARMS.Clear, MAIN.Cycle_Time, PARAMS.SF_Delay, SF006 );
F_CALC_SENSOR_NC ( N36_DI1_CH7_2 , ALARMS.Clear, MAIN.Cycle_Time, PARAMS.SF_Delay, SF007 );
F_CALC_SENSOR_NC ( N36_DI0_CH7_4 , ALARMS.Clear, MAIN.Cycle_Time, PARAMS.SF_Delay, SF008 );
F_CALC_SENSOR_NC ( N37_DI15_CH2_2, ALARMS.Clear, MAIN.Cycle_Time, PARAMS.SF_Delay, SF009 );

F_CALC_SENSOR_BAR ( N36_AI3_CH5_2 * 0.004, ALARMS.Clear,  P010 );
F_CALC_SENSOR_BAR ( N36_AI1_CH6_2 * 0.004, ALARMS.Clear,  P001 );
F_CALC_SENSOR_BAR ( N36_AI0_CH6_4 * 0.004, ALARMS.Clear,  P002 );
F_CALC_SENSOR_BAR ( N36_AI5_CH8_2 * 0.004, ALARMS.Clear,  P051 );
F_CALC_SENSOR_BAR ( N36_AI4_CH8_4 * 0.004, ALARMS.Clear,  P052 );

F_CALC_SENSOR_BAR ( N42_AI4_CH8_4 * 0.004, ALARMS.Clear,  P003 );

F_CALC_SENSOR_TEMP( N36_AI2_CH5_4 * 0.004, ALARMS.Clear, MAIN.Cycle_Time, S011 );

(*MF01 - Node22/42*)
(*F_CALC_SENSOR_NC ( N22_DI1_CH7_2, ALARMS.Clear, MAIN.Cycle_Time, 0.0, PTC101 );*)	(*New 20211008*)
(*F_CALC_SENSOR_NC ( N22_DI0_CH7_4, ALARMS.Clear, MAIN.Cycle_Time, 0.0, PTC102 );*)	(*New 20211008*)

F_CALC_SENSOR_TEMP( N21_AI5_CH8_2 * 0.001, ALARMS.Clear, MAIN.Cycle_Time, S101 );	(*New 20211008*)
F_CALC_SENSOR_TEMP( N21_AI4_CH8_4 * 0.001, ALARMS.Clear, MAIN.Cycle_Time, S102 );	(*New 20211008*)
F_CALC_SENSOR_TEMP( N42_AI5_CH8_2 * 0.004, ALARMS.Clear, MAIN.Cycle_Time, S100 );	(*New 20250117*)

F_CALC_SENSOR_BAR ( N42_AI1_CH6_2 * 0.004, ALARMS.Clear, P101 );
F_CALC_SENSOR_BAR ( N42_AI0_CH6_4 * 0.004, ALARMS.Clear, P103 );

F_CALC_SENSOR_NC ( N42_DI1_CH7_2, ALARMS.Clear, MAIN.Cycle_Time, PARAMS.SF_Delay, SF100 ); (*change to CH7 20250117*)


(*MF02 - Node34*)
F_CALC_SENSOR_BAR( N34_AI5_CH8_2 * 0.001, ALARMS.Clear,  P201 );

(*MF03 - Node43/44*)
F_CALC_SENSOR_BAR( N43_AI3_CH5_2 * 0.004, ALARMS.Clear,  P309 );
F_CALC_SENSOR_BAR( N43_AI2_CH5_4 * 0.004, ALARMS.Clear,  P311 );
F_CALC_SENSOR_BAR( N43_AI1_CH6_2 * 0.004, ALARMS.Clear,  P307 );

F_CALC_SENSOR_POS( N43_AI0_CH6_4 * 0.004, ALARMS.Clear, LS309 );
F_CALC_SENSOR_POS( N43_AI5_CH8_2 * 0.004, ALARMS.Clear, LS307 );
F_CALC_SENSOR_POS( N43_AI4_CH8_4 * 0.004, ALARMS.Clear, LS311 );

F_CALC_SENSOR_BAR( N44_AI3_CH5_2 * 0.004, ALARMS.Clear,  P301 );
F_CALC_SENSOR_BAR( N44_AI1_CH6_2 * 0.004, ALARMS.Clear,  P303 );
F_CALC_SENSOR_BAR( N44_AI5_CH8_2 * 0.004, ALARMS.Clear,  P305 );

